FOR aa := 0 TO iSafetyDiag_Anzahl_FbTwoHand DO
	(*	TwoHand (Taster) Diagnose		*)
	fbDiag_TwoHand[aa].stIn := Iarr_SafetyDiag_TwoHand[aa];
	fbDiag_TwoHand[aa]( );
	(*	Warnungen anzeigen	*)
	IF fbDiag_TwoHand[aa].bWarning THEN
		IEvent.Select(Tc_Events.TwinSafeEventClass.ErrorEvent)
			  .ArgSbInitWs(stTextListGlobal.stText_Safety.stText_Safety_FB_Error.wsName)
		  	  .ArgSbAppend(' | ')
			  .ArgSbAppendWsRaise(fbDiag_TwoHand[aa].stWarningText.wsName);
	END_IF
	(*	Error anzeigen	*)
	IF fbDiag_TwoHand[aa].bError THEN
		IEvent.Select(Tc_Events.TwinSafeEventClass.ErrorEvent)
			  .ArgSbInitWs(stTextListGlobal.stText_Safety.stText_Safety_FB_Error.wsName)
		  	  .ArgSbAppend(' | ')
			  .ArgSbAppendWsRaise(fbDiag_TwoHand[aa].stErrorText.wsName);
	END_IF
END_FOR

// EDM Diagnose
FOR aa := 0 TO iSafetyDiag_Anzahl_FbEDM DO
	(*	EDM FB Diagnose		*)
	fbDiag_EDM[aa].stIn := Iarr_SafetyDiag_EDM[aa];
	fbDiag_EDM[aa]( );
	(*	Error anzeigen	*)
	IF fbDiag_EDM[aa].bError THEN
		IEvent.Select(Tc_Events.TwinSafeEventClass.EdmErrorEvent)
			  .ArgSbInitWs(stTextListGlobal.stText_Safety.stText_Safety_FB_Error.wsName)
		  	  .ArgSbAppend(' | ')
			  .ArgSbAppendWsRaise(fbDiag_EDM[aa].stErrorText.wsName);
	END_IF
END_FOR


(*	Hardware	*)
FOR aa := 1 TO iSafety_Anzahl_EL69xx DO
	fbTwinSAFE_HW_Diag[aa].bEnable := Services.bPlcInitDone;
	fbTwinSAFE_HW_Diag[aa].stEcMasterAmsAdr := IO.stControlCabinetIO.stIn.stEtherCATMasterAmsAdr;
	fbTwinSAFE_HW_Diag[aa].nEcMasterDevId := IO.stControlCabinetIO.stIn.uiEcMasterDevId;
	fbTwinSAFE_HW_Diag[aa].nDeviceState := IO.stControlCabinetIO.stIn.eEtherCATDeviceState;
	fbTwinSAFE_HW_Diag[aa].dtNow := Statics.dtNow; // current system time
	fbTwinSAFE_HW_Diag[aa]();
	IF fbTwinSAFE_HW_Diag[aa].bError THEN
		IEvent.Select(Tc_Events.TwinSafeEventClass.HwErrorEvent)
		  	  .ArgSbInitWs(fbTwinSAFE_HW_Diag[aa].stErrorText.wsName)
		  	  .ArgSbAppendRaise(' | Safety Feedback Not-Halt');
	END_IF
END_FOR
END_METHOD

METHOD private M_DoorSequence : BOOL
VAR_INPUT
END_VAR
// Safe Gates

// A
fbSaftyDoors[0].sName := 'Tür Ofen A';
fbSaftyDoors[0].bAblaufGestoppt := Services.stGlobalModuleInfo.bStation_All_Stopped;
fbSaftyDoors[0].bFreigabeTuerEntriegeln := NOT fbSaftyDoors[0].bSAFE_AnforderungSchutzbereich_Ein;
fbSaftyDoors[0](stIO := Safety.arrSaftyDoors[0]);
IF fbSaftyDoors[0].bError THEN
	IEvent.Select(Tc_Events.TwinSafeEventClass.ErrorEvent)
		  .ArgSbInit('Türe A Fehler | ')
		  .ArgSbAppendWsRaise(fbSaftyDoors[0].stErrorText.wsName);
END_IF

// B
fbSaftyDoors[1].sName := 'Tür Ofen B';
fbSaftyDoors[1].bAblaufGestoppt := Services.stGlobalModuleInfo.bStation_All_Stopped;
fbSaftyDoors[1].bFreigabeTuerEntriegeln := NOT fbSaftyDoors[1].bSAFE_AnforderungSchutzbereich_Ein;
fbSaftyDoors[1](stIO := Safety.arrSaftyDoors[1]);
IF fbSaftyDoors[1].bError THEN
	IEvent.Select(Tc_Events.TwinSafeEventClass.ErrorEvent)
		  .ArgSbInit('Türe B Fehler | ')
		  .ArgSbAppendWsRaise(fbSaftyDoors[1].stErrorText.wsName);
END_IF

// reset
rtrigReset(CLK := HMI.stHmi.stIn.stSafety.bQuitSafety);
IF rtrigReset.Q THEN
	FOR ii := 0 TO 1 DO
		fbSaftyDoors[ii].M_Reset();
	END_FOR
END_IF

// request manual on request open door
bMachineRequestCycleStop := NOT (fbSaftyDoors[0].bFreigabeAblauf AND fbSaftyDoors[1].bFreigabeAblauf);
bMachineRequestStart := NOT bMachineRequestCycleStop AND (fbSaftyDoors[0].bStartAblauf OR fbSaftyDoors[1].bStartAblauf);
END_METHOD

METHOD private M_Edm : BOOL
VAR_INPUT
END_VAR
//ToDo: EDM
//bEdm_EmergencyStop:=TRUE;
//stEdm_State_Nothalt:= F_CreateDynText("Alle EDM Nothalt Signale OK", 0);	
//
//stIO.stOut.bSafety_EDM_OUT[E_EDM_Out.eEdmOut_Nothalt] := bEdm_EmergencyStop; //Nothalt

//stIO.stOut.bSafety_EDM_OUT[E_EDM_Out.eEdmOut_Modul1_Freigabeventil] := IO.st001_Modul_IO.stIn.bSignal_Modul1SafetyEdmVentilinsel;//AND IO.st001_Modul_IO.stIn.bSensor_Modul1PilotluftDs;//NOT stIO.stIn.bSafety_Aktor[E_Safety_Actor.eSafety_Actor_Freigabeventil_Area1];

//stIO.stOut.bSafety_EDM_OUT[E_EDM_Out.eEdmOut_Modul1_Rtt] := NOT SafetyArea2_Ok;

//EDM Check Meldungen

//fbEdmCheck[1].bEnable := TRUE;
//fbEdmCheck[1].bActor := stIO.stIn.bSAFE_ES_Ok;
//fbEdmCheck[1].bEdm := stIO.stOut.bSafety_EDM_OUT[E_EDM_Out.eEdmOut_Nothalt];
//fbEdmCheck[1].tActorOnEdmOffDelay := T#1S;
//fbEdmCheck[1].tActorOffEdmOnDelay := T#1S;
//fbEdmCheck[1]();
//IF fbEdmCheck[1].bEdmError THEN
//	fbEdmCheck[1].M_Reset();	
//																		
//	INotiHdl.M_SetNotification(F_CreateDynText("0",0),
//					stTextListGlobal.stText_NG_Safety, 							// Grp
//					stTextListGlobal.stText_Safety.stText_Safety_ES, 			// Text 1 (stTextListGlobal / F_CreateDynText("xxx",0))				 
//					F_CreateDynText("EDM Nothalt",0), 							// Text 2 (stTextListGlobal / F_CreateDynText("xxx",0))
//					stEdm_State_Nothalt,										// Text 3 (stTextListGlobal / F_CreateDynText("xxx",0))	
//					E_AlarmPriority.Warning,									// Priority
//					E_NotificationMode.eNotificationMode_Auto					// Notification mode (Autoreset or manually reset by user)
//					);										
//										
//END_IF
END_METHOD

METHOD private M_General : BOOL
VAR_INPUT
END_VAR
;
//Zustimm bereits in Safety ausgewertet mit Betriebsart
END_METHOD

METHOD INTERNAL M_Init : BOOL
VAR_INPUT
END_VAR
// init Safety stuff here...

// set up logger
ILog := Services.ILog;

// set up safety IOs
stIO REF= IO.stSafetyIO;

// set up event handler 
IEvent := Services.fbEventHandler;

//aSClearText[EN] := 'Safety init done.';
M_Init := TRUE;
END_METHOD

METHOD PRIVATE M_Mapping : BOOL
VAR_INPUT
END_VAR
stIO.stIn.bSAFE_DRIVES_STO := stIO.stIn.bSAFE_DRIVE_A_STO OR
								stIO.stIn.bSAFE_DRIVE_B_STO OR
								stIO.stIn.bSAFE_DRIVES_HG_STO;
								
//IO.stSafetyIO.stIn.bSAFE_Areas_Ok := IO.stSafetyIO.stIn. AND 
//									 IO.stSafetyIO.stIn.bSAFE_Area_Ok_ST20;
									 
									 
// machine stop from safety (ES/Door stop ramp)
bMachineRequestStop := NOT (stIO.stIn.bSAFE_ES_Ok AND
							IO.stSafetyIO.stIn.bSAFE_Areas_Ok );// AND
							//IO.stSafetyIO.stIn.bSAFE_Area_Ok_ST20);
END_METHOD

{attribute 'monitoring' := 'call'}
PROPERTY OpMode_Auto : BOOL
GET
OpMode_Auto := stIO.stIn.bSafe_OpMode_Auto;
END_GET
END_PROPERTY

{attribute 'monitoring' := 'call'}
PROPERTY OpMode_Manual : BOOL
GET
OpMode_Manual := stIO.stIn.bSafe_OpMode_Manual;
END_GET
END_PROPERTY

{attribute 'monitoring' := 'call'}
PROPERTY OpMode_Off : BOOL
GET
OpMode_Off := stIO.stIn.bSafe_OpMode_Off;
END_GET
END_PROPERTY

PROPERTY OpMode_Ruest : BOOL
GET
OpMode_Ruest := stIO.stIn.bSafe_OpMode_Ruest;
END_GET
END_PROPERTY

{attribute 'monitoring' := 'call'}
PROPERTY INTERNAL SafetyAreaOk_ST10 : BOOL
GET
SafetyAreaOk_ST10 := tofAreaOkST10.Q;
END_GET
END_PROPERTY

PROPERTY PUBLIC SafetyAreaOk_ST20 : BOOL
GET
SafetyAreaOk_ST20 := IO.stSafetyIO.stIn.bSAFE_Area_Ok_ST20;
END_GET
END_PROPERTY

{attribute 'monitoring' := 'call'}
PROPERTY PUBLIC SafetyOk : BOOL
GET // PUBLIC
SafetyOk := EmergencyStopOk AND IO.stSafetyIO.stIn.bSAFE_Areas_Ok;
END_GET
END_PROPERTY

END_PROGRAM

// ---- POUs/Safety/Components/Euchner_MGB2/FB_SafeDoorMGB2.TcPOU
FUNCTION_BLOCK FB_SafeDoorMGB2
VAR_IN_OUT
	// IO reference
	stIO 				: ST_MGB2_IO;
END_VAR
VAR_INPUT
	/// Name der Schutztuere
	sName								:STRING;
	
	bEnableSubModul_1					:BOOL := TRUE;
	bEnableSubModul_2					:BOOL := TRUE;
	
	/// Ablauf der Anlage gestoppt -> Freigabe zum Abschalten der Safety
	bAblaufGestoppt						:BOOL;
	
	/// Tuere entriegeln von Safety (Feedbacks)
	bFreigabeTuerEntriegeln				:BOOL;
END_VAR
VAR_OUTPUT
	/// Fehler
	bError								:BOOL;
	stErrorText							:ST_Text;
	
	/// Freigabe an Anlagenbereich zum Ausfueren der Abläufe
	bFreigabeAblauf							:BOOL;
	
	/// Anforderung an Safety für Sicherheit
	bSAFE_AnforderungSchutzbereich_Ein		:BOOL;
END_VAR
VAR
	stInMgb						: ST_Euchner_MGB2_IN;
	stOutMgb					: ST_Euchner_MGB2_Out;
	stInMsm						: ST_Euchner_MSM_IN;
	stOutMsm					: ST_Euchner_MSM_Out;
	stInMsmConfirm				: ST_Euchner_MSM_DA_IN;
	stOutMsmConfirm				: ST_Euchner_MSM_DA_Out;
	
	bReset,
	bStarting,
	bLockDoorRequest,
	bOpenDoorRequest			:BOOL;
	fbTaAnforderung				:FB_TON_RMTH;
	fbTaQuittieren				:FB_TON_RMTH;
	fbSafetyOk					:FB_TON_RMTH;
	tonReset					: TON;
END_VAR

M_Mapping();
M_Supervision();

// Timer, Flanken
fbTaAnforderung(IN := stInMsm.bSM_I_S2, PT:= T#50MS);		// stIO.stIn.bTa_Gelb_S2
fbTaQuittieren(IN := stInMsm.bSM_I_S3, PT:= T#50MS);		// stIO.stIn.bTa_Weiss_S3

stOutMsm.bSM_O_H1 := FALSE;
stOutMsm.bSM_O_H2 := FALSE;
stOutMsm.bSM_O_H3 := FALSE;

tonReset.IN := bReset;
tonReset.PT := T#150MS;
tonReset();
IF tonReset.Q THEN
	bReset := FALSE;
END_IF
stOutMgb.bLM_ACK_ER := stOutMgb.bLM_ACK_G := bReset;
stOutMgb.bLM_ACK_G := stOutMgb.bLM_ACK_G := bReset;

(*	Funktion OK	*)
IF NOT bError THEN

	// mapp ES button to led
	IF NOT stInMsm.bSM_I_S1 THEN
		stOutMsm.bSM_O_H1 := Statics.stPulse.bToggle500ms; 
	ELSE
		stOutMsm.bSM_O_H1 := FALSE;
	END_IF

	//---------------------------- Open ---------------------------------
	// Anforderung Tuere oeffnen
	IF fbTaAnforderung.Qr OR bOpenDoorRequest THEN
		bOpenDoorRequest := FALSE;
		bFreigabeAblauf := FALSE;
		bStarting := FALSE;
	END_IF
	// Safety abschalten
	IF NOT bFreigabeAblauf AND bAblaufGestoppt AND 	// Abläufe sind gestoppt in dem Bereich
	NOT bStarting THEN
		bSAFE_AnforderungSchutzbereich_Ein := FALSE;		// Abschalten in Safety
	END_IF
	
	// Rückmeldung von Safety das entriegelt werden darf
	IF NOT bSAFE_AnforderungSchutzbereich_Ein AND 
	bFreigabeTuerEntriegeln AND NOT bStarting THEN
		stOutMgb.bLM_O_CL := TRUE; // entriegeln	
	END_IF
	
	
	// Signal LED - Gelb
	IF bStarting THEN
		stOutMsm.bSM_O_H2 := FALSE;	
	ELSIF NOT bFreigabeAblauf AND NOT bFreigabeTuerEntriegeln THEN
		stOutMsm.bSM_O_H2 := Statics.stPulse.bToggle500ms;
	ELSIF NOT stIO.bSAFE_DoorSafetyOk THEN
		stOutMsm.bSM_O_H2 := TRUE;
	ELSE
		stOutMsm.bSM_O_H2 := FALSE;
	END_IF
	
	
	//---------------------------- Close + Start --------------------------
	// Tuere quittieren (geschlossen und verriegeln) -> fallende Flanke
	IF fbTaQuittieren.Qf OR bLockDoorRequest THEN
		bLockDoorRequest := FALSE;
		IF stInMgb.bLM_I_SK AND stInMgb.bLM_I_OL THEN	// stIO.stIn.bMeldungRiegelzunge_OT   stInMgb.bLM_I_SK AND stInMgb.bLM_I_OL
			stOutMgb.bLM_O_CL := FALSE; // verriegeln
			bSAFE_AnforderungSchutzbereich_Ein := TRUE;	// Safety Ein
			bStarting := TRUE;
		END_IF
	END_IF
	
	fbSafetyOk(IN := stIO.bSAFE_DoorSafetyOk, PT := T#200MS);
	IF bStarting THEN
		IF fbSafetyOk.Q THEN
			bFreigabeAblauf := TRUE;
			bStarting := FALSE;
		END_IF
	END_IF
	
	// Signal LED - Weiss
	IF stIO.bSAFE_DoorSafetyOk THEN
		stOutMsm.bSM_O_H3 := TRUE;
	ELSIF bStarting THEN
		stOutMsm.bSM_O_H3 := Statics.stPulse.bToggle500ms;
	ELSIF stInMgb.bLM_I_OT THEN		// stIO.stIn.bMeldungRiegelzunge_OT
		stOutMsm.bSM_O_H3 := Statics.stPulse.bToggle1000ms;
	ELSE
		stOutMsm.bSM_O_H3 := FALSE;
	END_IF
	
// 
// ERROR
ELSE

	stOutMsm.bSM_O_H1 := Statics.stPulse.bToggle500ms;
	stOutMsm.bSM_O_H2 := Statics.stPulse.bToggle500ms;
	stOutMsm.bSM_O_H3 := Statics.stPulse.bToggle500ms;

	stOutMgb.bLM_O_CL := TRUE;
	IF stInMsm.bSM_I_S2 OR stInMsm.bSM_I_S3 THEN
		bReset := TRUE;
	END_IF
	IF stInMsm.bSM_I_S2 AND stInMgb.bLM_I_SK AND stInMgb.bLM_I_OL THEN
		stOutMgb.bLM_O_CL := FALSE;
	ELSIF stInMsm.bSM_I_S3 THEN	(*AND bEnable*)
		stOutMgb.bLM_O_CL := TRUE;
	END_IF
	
END_IF

stIO.bSAFE_UnlockDoor := stOutMgb.bLM_O_CL;

METHOD PRIVATE M_Error : BOOL
VAR_INPUT
	stError: ST_Text;
END_VAR
bError	:=TRUE;
stErrorText	:= stError;
END_METHOD

METHOD M_LockDoor : BOOL
VAR_INPUT
END_VAR
//IF stInMgb.bLM_I_OT THEN
	bLockDoorRequest := TRUE;	
//END_IF
END_METHOD

METHOD PRIVATE M_Mapping : BOOL
//mgb mapping in
stInMgb.bLM_D_RUN := 	stIO.stHwInMgb.nByte0.0;
stInMgb.bLM_I_SK := 	stIO.stHwInMgb.nByte0.1;
stInMgb.bLM_E_SM1 := 	stIO.stHwInMgb.nByte0.2;
stInMgb.bLM_E_SM2 := 	stIO.stHwInMgb.nByte0.3;
stInMgb.bLM_E_ER := 	stIO.stHwInMgb.nByte0.4;
stInMgb.bLM_E_G := 		stIO.stHwInMgb.nByte0.5;
stInMgb.bLM_I_OD := 	stIO.stHwInMgb.nByte0.6;
stInMgb.bLM_I_OT := 	stIO.stHwInMgb.nByte0.7;
stInMgb.bLM_I_OL := 	stIO.stHwInMgb.nByte1.0;

//mgb mapping out
stIO.stHwOutMgb.nByte0.0 := stOutMgb.bLM_O_CL;
stIO.stHwOutMgb.nByte0.1 := stOutMgb.bLM_ACK_ER;
stIO.stHwOutMgb.nByte0.2 := stOutMgb.bLM_ACK_G;

//msm mapping in
stInMsm.bSM_I_S1 := 	stIO.stHwInMsm.nByte0.0;
stInMsm.bSM_I_S2 := 	stIO.stHwInMsm.nByte0.1;
stInMsm.bSM_I_S3 := 	stIO.stHwInMsm.nByte0.2;
stInMsm.bSM_E_S1 := 	stIO.stHwInMsm.nByte0.5;

stInMsmConfirm.bSM_I_X3 := 	stIO.stHwInMsmConfirm.nByte0.0;	// Zustimm
stInMsmConfirm.bSM_I_T1 := 	stIO.stHwInMsmConfirm.nByte0.2;	// Minus
stInMsmConfirm.bSM_I_T2 := 	stIO.stHwInMsmConfirm.nByte0.1; // Plus
stInMsmConfirm.bSM_E_X3 := 	stIO.stHwInMsmConfirm.nByte0.5;

//msm mapping out
stIO.stHwOutMsm.nByte0.0 := stOutMsm.bSM_O_H1;
stIO.stHwOutMsm.nByte0.1 := stOutMsm.bSM_O_H2;
stIO.stHwOutMsm.nByte0.2 := stOutMsm.bSM_O_H3;
stIO.stHwOutMsm.nByte0.3 := stOutMsm.bSM_O_H1_B;
stIO.stHwOutMsm.nByte0.4 := stOutMsm.bSM_O_H2_B;
stIO.stHwOutMsm.nByte0.5 := stOutMsm.bSM_O_H3_B;

stIO.stHwOutMsmConfirm.nByte0.0 := stOutMsmConfirm.bSM_O_L2;
stIO.stHwOutMsmConfirm.nByte0.1 := stOutMsmConfirm.bSM_O_L1;
stIO.stHwOutMsmConfirm.nByte0.3 := stOutMsmConfirm.bSM_O_L2_B;
stIO.stHwOutMsmConfirm.nByte0.4 := stOutMsmConfirm.bSM_O_L1_B;
END_METHOD

METHOD M_OpenDoor : BOOL
VAR_INPUT
END_VAR
bOpenDoorRequest := TRUE;
END_METHOD

METHOD M_Reset : BOOL
bReset	:= TRUE;
bError	:= FALSE;
MEMSET(ADR(stErrorText),0,SIZEOF(stErrorText));
END_METHOD

METHOD PRIVATE M_Supervision : BOOL
IF stInMgb.bLM_E_SM1 AND bEnableSubModul_1 AND FALSE THEN
	M_Error(F_CreateDynTextEx(0, "Safety_MGB2_ErrBit_Submod1", "MGB2 - Fehlermeldebit für Submodul 1")); 	
ELSIF stInMgb.bLM_E_SM2 AND bEnableSubModul_2 THEN
	M_Error(F_CreateDynTextEx(0, "Safety_MGB2_ErrBit_Submod2", "MGB2 - Fehlermeldebit für Submodul 2"));	
ELSIF stInMgb.bLM_E_ER THEN
	M_Error(F_CreateDynTextEx(0, "Safety_MGB2_ErrBit_EscapeUnlock", "MGB2 - für Fluchtentriegelung"));	
ELSIF stInMgb.bLM_E_G THEN
	M_Error(F_CreateDynTextEx(0, "Safety_MGB2_ErrBit_ModError", "MGB2 - allgemeiner Modulfehler"));
ELSIF stInMsm.bSM_E_S1 THEN
	M_Error(F_CreateDynTextEx(0, "Safety_MSM_ErrBit_Sx", "MSM - Fehler"));
END_IF
END_METHOD

END_FUNCTION_BLOCK

// ---- POUs/HMI/Utilities/DynTxt/F_CreateDynTextEx.TcPOU
FUNCTION F_CreateDynTextEx : ST_Text
VAR_INPUT
	nNameId		: INT;		//example simatic hmi
	wsNameId	: WSTRING;	//standard name
	wsName		: WSTRING;	//standard name
END_VAR

F_CreateDynTextEx.nNameId := nNameId;
F_CreateDynTextEx.wsNameId := wsNameId;
F_CreateDynTextEx.wsName := wsName;

END_FUNCTION

// ---- POUs/Safety/Components/SafetyDoor/FB_SafetyDoor.TcPOU
FUNCTION_BLOCK FB_SafetyDoor
VAR_IN_OUT
	// IO reference
	stIO 				: ST_SafetyDoor_IO;
END_VAR
VAR_INPUT
	/// Name der Schutztuere
	sName								:STRING;
	
	bEnableSubModul_1					:BOOL := TRUE;
	bEnableSubModul_2					:BOOL := TRUE;
	
	/// Ablauf der Anlage gestoppt -> Freigabe zum Abschalten der Safety
	bAblaufGestoppt						:BOOL;
	
	/// Tuere entriegeln von Safety (Feedbacks)
	bFreigabeTuerEntriegeln				:BOOL;
END_VAR
VAR_OUTPUT
	/// Fehler
	bError								:BOOL;
	stErrorText							:ST_Text;
	
	/// Freigabe an Anlagenbereich zum Ausfueren der Abläufe
	bFreigabeAblauf,
	bStartAblauf 						: BOOL;
	
	/// Anforderung an Safety für Sicherheit
	bSAFE_AnforderungSchutzbereich_Ein	: BOOL;
END_VAR
VAR
	stIn					: ST_SafetyDoor_IN;
	stOut					: ST_SafetyDoor_OUT;
	
	bReset,
	bStarting				: BOOL;
	fbTaAnforderung			:FB_TON_RMTH;
	fbTaLock				:FB_TON_RMTH;
	fbTaStart				:FB_TON_RMTH;
	fbSafetyOk				:FB_TON_RMTH;
	tonReset, tonDelay		: TON;
	nStep					: INT;
END_VAR

M_Mapping();

// Timer, Flanken
fbTaAnforderung(IN := stIn.bRequestButton, PT:= T#50MS);	//Blau	
fbTaLock(IN := stIn.bLockButton, PT:= T#50MS);				//Gelb 
fbTaStart(IN := stIn.bStartButton, PT:= T#50MS);			//Grün 
fbSafetyOk(IN := stIn.tsSafe, PT := T#200MS);				//Safety

bStartAblauf := FALSE;

tonReset.IN := bReset;
tonReset.PT := T#150MS;
tonReset();
IF tonReset.Q THEN
	bReset := FALSE;
END_IF
//stOut.tsRestart := bReset;

(*	Funktion OK	*)
IF NOT bError THEN

	//---------------------------- Open ---------------------------------
	// Anforderung Tuere oeffnen
	IF fbTaAnforderung.Qr THEN
		bFreigabeAblauf := FALSE;
		bStarting := FALSE;
	END_IF
	
	// Safety abschalten
	IF NOT bFreigabeAblauf AND bAblaufGestoppt AND 	 // Abläufe sind gestoppt in dem Bereich
	NOT bStarting THEN
		bSAFE_AnforderungSchutzbereich_Ein := FALSE; // Abschalten in Safety
	END_IF
	
	// Rückmeldung von Safety das entriegelt werden darf
	IF fbTaLock.Qf THEN
		//---------------------------- Close + Start --------------------------
		// Tuere quittieren (geschlossen und verriegeln) -> fallende Flanke
		IF NOT stOut.tsLockCmd THEN
			nStep := 10; // lock
		ELSE
			nStep := 100; // open
		END_IF
	END_IF
	
	IF fbTaStart.Qf OR bStarting THEN
		IF fbSafetyOk.Q THEN
			bFreigabeAblauf := TRUE;
			bStartAblauf := TRUE;
			bStarting := FALSE;
		END_IF
	END_IF
	
	
	
	//---------------------------- Lights --------------------------	
	// Signal LED - Grün/Gelb	
	IF Services.stGlobalModuleInfo.bStation_All_Auto THEN
		IF Services.stGlobalModuleInfo.bStation_All_Started THEN
			stOut.bStartLight := TRUE;
			stOut.bStopLight := FALSE;
		ELSIF Services.stGlobalModuleInfo.bStation_All_Stopped THEN
			stOut.bStartLight := FALSE;
			stOut.bStopLight := TRUE;
		ELSIF bFreigabeAblauf THEN
			stOut.bStartLight := Statics.stPulse.bToggle500ms;
			stOut.bStopLight := Statics.stPulse.bToggle500ms;
		END_IF
	ELSE
		stOut.bStartLight := FALSE;
		stOut.bStopLight := FALSE;
	END_IF	
	
	// Signal LED - Gelb
	stOut.bLockLight := NOT stIn.tsOpen;	
// 
// ERROR
ELSE

	stOut.bLockLight := Statics.stPulse.bToggle500ms;
	stOut.bStopLight := Statics.stPulse.bToggle500ms;
	stOut.tsLockCmd := FALSE;
	
END_IF

tonDelay();
CASE nStep OF
	0: // idle
		IF stIn.tsOpen THEN
			nStep := 10;
		END_IF
	
	10: // lock
		IF stIn.tsSafe THEN
			nStep := 30;
		ELSE
			tonDelay(IN := FALSE);
			stOut.tsRestart := TRUE;
			nStep := 20;
		END_IF
		
	20: // restart door fb (delay)
		tonDelay(IN := TRUE, PT := T#300MS);
		IF tonDelay.Q THEN
			tonDelay(IN := FALSE);
			stOut.tsRestart := FALSE;
			nStep := 10;
		END_IF
		
	30: // lock
		stOut.tsLockCmd := TRUE; // verriegeln
		bSAFE_AnforderungSchutzbereich_Ein := TRUE;	// Safety Ein
		bStarting := TRUE;
		nStep := 0;
		
	100: // open
		bFreigabeAblauf := FALSE;
		bStarting := FALSE;
	
		IF NOT bSAFE_AnforderungSchutzbereich_Ein AND 
		bFreigabeTuerEntriegeln AND NOT bStarting THEN
			stOut.tsLockCmd := FALSE; // entriegeln
			nStep := 0;
		END_IF
		
		
END_CASE

METHOD PRIVATE M_Error : BOOL
VAR_INPUT
	stError: ST_Text;
END_VAR
bError	:=TRUE;
stErrorText	:= stError;
END_METHOD

METHOD PRIVATE M_Mapping : BOOL
//mgb mapping in
stIn := stIO.stHwIn;

stOut.tsLocked := stIn.bLocked;

stIO.stHwOut := stOut;
END_METHOD

METHOD M_Reset : BOOL
bReset	:= TRUE;
bError	:= FALSE;
MEMSET(ADR(stErrorText),0,SIZEOF(stErrorText));
END_METHOD

END_FUNCTION_BLOCK

// ---- POUs/HMI/Utilities/DynTxt/F_CreateDynText.TcPOU
FUNCTION F_CreateDynText : ST_Text
VAR_INPUT
	wsName		: WSTRING;	//standard name
	nNameId		: INT;		//example simatic hmi
END_VAR
VAR
END_VAR

F_CreateDynText.wsName := wsName;
F_CreateDynText.wsNameId := wsName;
F_CreateDynText.nNameId := nNameId;

END_FUNCTION

// ---- POUs/HMI/P_HMI_Controller.TcPOU
/// HMI access provider (host for sub hmi provider)
PROGRAM INTERNAL P_HMI_Controller
VAR_OUTPUT	
	// default items from HMI to module & stations
	aStHmiToModule	: ARRAY[0..E_Module.eModule_nMaxIdx] OF ST_DefaultHmiToPlc;
	aStHmiToStation	: ARRAY[0..E_Station.eStation_nMaxIdx] OF ST_DefaultHmiToPlc;
	bLedTest 		: BOOL;
END_VAR
VAR
	stHmiBaseOut	: ST_HMI_BASE_OUT;
	IEvent			: I_EventHandler;
	aiHmiProvider	: ARRAY[0..E_HMI_PROVIDER.eHmiProvider_nMaxIdx] OF ITF_HMI_PROVIDER;

	// default trigger
	aFbProviderRequestTrigger	: ARRAY[0..E_HMI_PROVIDER.eHmiProvider_nMaxIdx] OF FB_ProviderRequestTrigger;
	
	aFbTrigHmiToModule			: ARRAY[0..eModule_nMaxIdx] OF FB_HmiBaseControlTrigger;
	aFbTrigHmiToStation			: ARRAY[0..eStation_nMaxIdx] OF FB_HmiBaseControlTrigger;
			
	/// private variabe
	ii							: INT;
	stHmiInEmpty 				: ST_HMI_IN;	
	
	sChanges					: T_MaxString;
	fbSettingsHandling 			: FB_SettingsHandling;
	fbMonitoringHandling		: FB_MonitoringHandling;
	
	tonUserLevelLogOut				: TON;
	rTrigUserManagmentLogIn,
	rTrigUserManagmentLogOut,
	rTrigUserManagmentSubmit		: R_TRIG;	
	fTrigUserManagmentSubmit		: F_TRIG;
	rTrigUserManagmentDelete		: R_TRIG;
	
	nUserManagemenetColumnIdx_Old	: UINT;
	nUserManagemenetRowIdx_Old		: UINT;
	
	sUserLevelLastUser				: STRING;
	stAxisManagerDummy 				: ST_AxisManager;
END_VAR
VAR PERSISTENT
	// user data
	iUserLevel					: INT;	(*user level 0 = none 1= Operator 2 = Plant Manager 3 = maintenance 4 = reserve 5= admin 6= programmer*)
	stUserLevel					: ARRAY [0..20] OF ST_User_Management;
	bPasswordSave				: BOOL;
END_VAR

///
/// HMI access provider
/// 

// build general HMI out
M_PlcToHmi();

// init summary IN (resets combined or-signals)
stHMI.stIn := stHmiInEmpty;

// loop provider, run & chk control requests
FOR ii := 0 TO E_HMI_PROVIDER.eHmiProvider_nMaxIdx DO
	IF aiHmiProvider[ii] = 0 THEN CONTINUE;	END_IF
	
	M_PlcToProvider(aiHmiProvider[ii]);
	aiHmiProvider[ii].M_Run();
	IF aiHmiProvider[ii].Mute THEN CONTINUE; END_IF
	M_ProviderToPlc(aiHmiProvider[ii], aFbProviderRequestTrigger[ii]);
END_FOR

bLedTest := stHmi.stIn.stSpecial.stButton_LedTest.bClick;

// build module & station signals
M_HmiToModules();
M_HmiToStations();

// user mgmt --> switched to Beckhoff HMI UserMgmt
HMI.eUserLevel := HMI.stHmiTc3.stIn.stUserMgmt.iHmiUserLevel;
//M_UserManagement();
M_AxisManagement();

// reset
IF stHmi.stIn.stMain.stButton_Reset.bClick THEN
	M_Reset();
END_IF

METHOD PRIVATE M_AddSystemInfo : BOOL
VAR
	idx : INT;
END_VAR
// add/update system infos
idx := 0;
M_UpdateSystemInfo('App.ProjectName', Statics.stPlcSystemInfo.stPlcAppSystemInfo.ProjectName, idx);
M_UpdateSystemInfo('Software Version', stLibVersion_PLC.sVersion, idx);
M_UpdateSystemInfo('Safety Device Serial', UDINT_TO_STRING(IO.stSafetyIO.stIn.nSerialNumber), idx);
M_UpdateSystemInfo('Safety Project CRC', WORD_TO_STRING(IO.stSafetyIO.stIn.nProjectCrc), idx);
M_UpdateSystemInfo('', '', idx);
M_UpdateSystemInfo('App.AppName', Statics.stPlcSystemInfo.stPlcAppSystemInfo.AppName, idx);
M_UpdateSystemInfo('App.AppTimestamp', DT_TO_STRING(Statics.stPlcSystemInfo.stPlcAppSystemInfo.AppTimestamp), idx);
M_UpdateSystemInfo('App.AdsPort', UDINT_TO_STRING(Statics.stPlcSystemInfo.stPlcAppSystemInfo.AdsPort), idx);
M_UpdateSystemInfo('App.ObjId', UDINT_TO_STRING(Statics.stPlcSystemInfo.stPlcAppSystemInfo.ObjId), idx);
M_UpdateSystemInfo('App.TaskCnt', UDINT_TO_STRING(Statics.stPlcSystemInfo.stPlcAppSystemInfo.TaskCnt), idx);
M_UpdateSystemInfo('App.OnlineChangeCnt', UDINT_TO_STRING(Statics.stPlcSystemInfo.stPlcAppSystemInfo.OnlineChangeCnt), idx);
M_UpdateSystemInfo('App.Flags', DWORD_TO_STRING(Statics.stPlcSystemInfo.stPlcAppSystemInfo.Flags), idx);
M_UpdateSystemInfo('App.BootDataLoaded', BOOL_TO_STRING(Statics.stPlcSystemInfo.stPlcAppSystemInfo.BootDataLoaded), idx);
M_UpdateSystemInfo('App.OldBootData', BOOL_TO_STRING(Statics.stPlcSystemInfo.stPlcAppSystemInfo.OldBootData), idx);
M_UpdateSystemInfo('App.KeepOutputsOnBP', BOOL_TO_STRING(Statics.stPlcSystemInfo.stPlcAppSystemInfo.KeepOutputsOnBP), idx);
M_UpdateSystemInfo('App.ShutdownInProgress',  BOOL_TO_STRING(Statics.stPlcSystemInfo.stPlcAppSystemInfo.ShutdownInProgress), idx);
M_UpdateSystemInfo('App.LicensesPending',  BOOL_TO_STRING(Statics.stPlcSystemInfo.stPlcAppSystemInfo.LicensesPending), idx);
M_UpdateSystemInfo('App.BSODOccured',  BOOL_TO_STRING(Statics.stPlcSystemInfo.stPlcAppSystemInfo.BSODOccured), idx);	 
//M_AddSystemInfo('App.TComSrvPtr', Statics.stPlcSystemInfo.stPlcAppSystemInfo.TComSrvPtr, idx); 
M_UpdateSystemInfo('Task.TaskName', Statics.stPlcSystemInfo.stPlcTaskSystemInfo.TaskName, idx);
M_UpdateSystemInfo('Task.AdsPort', UINT_TO_STRING(Statics.stPlcSystemInfo.stPlcTaskSystemInfo.AdsPort), idx);
M_UpdateSystemInfo('Task.Priority', UINT_TO_STRING(Statics.stPlcSystemInfo.stPlcTaskSystemInfo.Priority), idx);
M_UpdateSystemInfo('Task.CycleTime', Concat2x(F_LRealToStringEx(Statics.stPlcSystemInfo.fCycleTime * 1E3, 0), ' ms, '), idx);
M_UpdateSystemInfo('Task.LastExecTime', Concat2x(F_LRealToStringEx(Statics.stPlcSystemInfo.fLastExecTime * 1E6, 1), ' µs'), idx);
M_UpdateSystemInfo('Task.CycleCount',UDINT_TO_STRING(Statics.stPlcSystemInfo.stPlcTaskSystemInfo.CycleCount), idx);
M_UpdateSystemInfo('Task.DcTaskTime', LINT_TO_STRING(Statics.stPlcSystemInfo.stPlcTaskSystemInfo.DcTaskTime), idx);
M_UpdateSystemInfo('Task.FirstCycle', BOOL_TO_STRING(Statics.stPlcSystemInfo.stPlcTaskSystemInfo.FirstCycle), idx);
M_UpdateSystemInfo('Task.CycleTimeExceeded', BOOL_TO_STRING(Statics.stPlcSystemInfo.stPlcTaskSystemInfo.CycleTimeExceeded), idx);
M_UpdateSystemInfo('Task.InCallAfterOutputUpdate', BOOL_TO_STRING(Statics.stPlcSystemInfo.stPlcTaskSystemInfo.InCallAfterOutputUpdate), idx);
M_UpdateSystemInfo('Task.RTViolation', BOOL_TO_STRING(Statics.stPlcSystemInfo.stPlcTaskSystemInfo.RTViolation), idx);
END_METHOD

METHOD M_AxisManagement : INT
VAR_INPUT
	
END_VAR
IF NOT Services.bPlcInitDone THEN
	RETURN;
END_IF

HMI.stHmiInOut.stHmiAxisManager.bEnableAxisMgr := P_Safety.OpMode_Off;

CASE HMI.stHmiInOut.stHmiAxisManager.eAxis OF
	E_Axis.eAxis_OvenA: HMI.stHmiInOut.stHmiAxisManager.stAxisManager REF= fbSt010OvenA.fbAxisUi.stAxisManager;
	E_Axis.eAxis_OvenB: HMI.stHmiInOut.stHmiAxisManager.stAxisManager REF= fbSt020OvenB.fbAxisUi.stAxisManager;
	
	E_Axis.eAxis_Handling_X: HMI.stHmiInOut.stHmiAxisManager.stAxisManager REF= fbSt030Handling.fbAxisXUi.stAxisManager;
	E_Axis.eAxis_Handling_Y: HMI.stHmiInOut.stHmiAxisManager.stAxisManager REF= fbSt030Handling.fbAxisYUi.stAxisManager;
	E_Axis.eAxis_Handling_Z: HMI.stHmiInOut.stHmiAxisManager.stAxisManager REF= fbSt030Handling.fbAxisZUi.stAxisManager;
	
	ELSE
		;//HMI.stHmiInOut.stHmiAxisManager.stAxisManager REF= fbModul001.fbAxisVmUi.stAxisManager;
END_CASE
END_METHOD

METHOD PRIVATE M_CombineCommonSignals : BOOL
VAR_IN_OUT
	stCtrlSum : ST_HMI_BASE_CONTROL_IN;
	stCtrlPrv : ST_HMI_BASE_CONTROL_IN;
END_VAR
F_OR_REF(stCtrlSum.stButton_Start.bClick, 		stCtrlPrv.stButton_Start.bClick);
F_OR_REF(stCtrlSum.stButton_CycleStop.bClick,	stCtrlPrv.stButton_CycleStop.bClick);
F_OR_REF(stCtrlSum.stButton_Stop.bClick, 		stCtrlPrv.stButton_Stop.bClick);
F_OR_REF(stCtrlSum.stButton_Home.bClick, 		stCtrlPrv.stButton_Home.bClick);
F_OR_REF(stCtrlSum.stButton_Step.bClick, 		stCtrlPrv.stButton_Step.bClick);
F_OR_REF(stCtrlSum.stButton_Reset.bClick, 		stCtrlPrv.stButton_Reset.bClick);
F_OR_REF(stCtrlSum.stButton_OPM_Auto.bClick,	stCtrlPrv.stButton_OPM_Auto.bClick);
F_OR_REF(stCtrlSum.stButton_OPM_Step.bClick,	stCtrlPrv.stButton_OPM_Step.bClick);
F_OR_REF(stCtrlSum.stButton_OPM_Manual.bClick,	stCtrlPrv.stButton_OPM_Manual.bClick);

M_CombineCommonSignals := TRUE;
END_METHOD

METHOD PRIVATE M_HmiToModules : BOOL
VAR
	ii	: INT;
END_VAR
// loop modules, default HMI to module (start, stop, reset, OpModes,...)
FOR ii := 0 TO E_Module.eModule_nMaxIdx DO
	// run only for valid modules
	IF P_Plant.aIModule[ii] = 0 THEN
		CONTINUE;
	END_IF

	aFbTrigHmiToModule[ii].stHmiToPlcIn.bStart := 			stHmi.stIn.arrStModule[ii].stButton_Start.bClick OR 
															stHmi.stIn.stMain.stButton_Start.bClick;
															
	aFbTrigHmiToModule[ii].stHmiToPlcIn.bStop := 			stHmi.stIn.arrStModule[ii].stButton_CycleStop.bClick OR 
															stHmi.stIn.stMain.stButton_Stop.bClick;
															
	aFbTrigHmiToModule[ii].stHmiToPlcIn.bFastStop := 		stHmi.stIn.arrStModule[ii].stButton_Stop.bClick OR 
															stHmi.stIn.stMain.stButton_CycleStop.bClick;
															
	aFbTrigHmiToModule[ii].stHmiToPlcIn.bReset := 			stHmi.stIn.arrStModule[ii].stButton_Reset.bClick OR 
															stHmi.stIn.stMain.stButton_Reset.bClick;

	aFbTrigHmiToModule[ii].stHmiToPlcIn.bStep := 			stHmi.stIn.arrStModule[ii].stButton_Step.bClick OR 
															stHmi.stIn.stMain.stButton_Step.bClick; 
															
	aFbTrigHmiToModule[ii].stHmiToPlcIn.bHome := 			stHmi.stIn.arrStModule[ii].stButton_Home.bClick OR 
															stHmi.stIn.stMain.stButton_Home.bClick; 
															
	aFbTrigHmiToModule[ii].stHmiToPlcIn.bOpModeManual := 	stHmi.stIn.arrStModule[ii].stButton_OPM_Manual.bClick OR 
															stHmi.stIn.stMain.stButton_OPM_Manual.bClick; 
															
	aFbTrigHmiToModule[ii].stHmiToPlcIn.bOpModeAuto := 		stHmi.stIn.arrStModule[ii].stButton_OPM_Auto.bClick OR 
															stHmi.stIn.stMain.stButton_OPM_Auto.bClick; 
															
	aFbTrigHmiToModule[ii].stHmiToPlcIn.bOpModeStep := 		stHmi.stIn.arrStModule[ii].stButton_OPM_Step.bClick OR 
															stHmi.stIn.stMain.stButton_OPM_Step.bClick;

	IF P_Safety.OpMode_Auto THEN
		aFbTrigHmiToModule[ii].stHmiToPlcIn.eSafetyOpMode := E_OpMode.eOpMode_auto;
	ELSIF P_Safety.OpMode_Manual THEN		
		aFbTrigHmiToModule[ii].stHmiToPlcIn.eSafetyOpMode := E_OpMode.eOpMode_manual;
//		ELSIF P_Safety.Betriebsart_Ruest THEN		
//			aFbTrigHmiToModule[ii].stHmiToPlcIn.eSafetyOpMode := E_OpMode.eOpMode_manual;
	ELSIF P_Safety.OpMode_Off THEN
		aFbTrigHmiToModule[ii].stHmiToPlcIn.eSafetyOpMode := E_OpMode.eOpMode_off;
	ELSE
		aFbTrigHmiToModule[ii].stHmiToPlcIn.eSafetyOpMode := E_OpMode.eOpMode_off;
	END_IF

	aFbTrigHmiToModule[ii](stHmiToPlcOut := aStHmiToModule[ii]);
END_FOR
END_METHOD

METHOD PRIVATE M_HmiToStations : BOOL
VAR
	ii	: INT;
	ISt	: IStation;
END_VAR
// loop stations, default HMI to mostationdule (start, stop, reset, OpModes,...)
FOR ii := 0 TO E_Station.eStation_nMaxIdx DO
	// run only for valid stations
	IF P_Plant.aIStaton[ii] = 0 THEN
		CONTINUE;
	END_IF

	ISt := P_Plant.aIStaton[ii];
	aFbTrigHmiToStation[ii].stHmiToPlcIn.bStart := 			stHmi.stIn.arrStStation[ii].stButton_Start.bClick OR 
															//to start all stations of the module:
															//stHmi.stIn.arrStModule[ISt.Parent].stButton_Start.bClick OR 
															stHmi.stIn.stMain.stButton_Start.bClick;
															
	aFbTrigHmiToStation[ii].stHmiToPlcIn.bStop := 			stHmi.stIn.arrStStation[ii].stButton_CycleStop.bClick OR 
															//stHmi.stIn.arrStModule[ISt.Parent].stButton_CycleStop.bClick OR 
															stHmi.stIn.stMain.stButton_Stop.bClick;
															
	aFbTrigHmiToStation[ii].stHmiToPlcIn.bFastStop := 		stHmi.stIn.arrStStation[ii].stButton_Stop.bClick OR 
															//stHmi.stIn.arrStModule[ISt.Parent].stButton_Stop.bClick OR 
															stHmi.stIn.stMain.stButton_CycleStop.bClick;
															
	aFbTrigHmiToStation[ii].stHmiToPlcIn.bReset := 			stHmi.stIn.arrStStation[ii].stButton_Reset.bClick OR 
															//stHmi.stIn.arrStModule[ISt.Parent].stButton_Reset.bClick OR 
															stHmi.stIn.stMain.stButton_Reset.bClick;

	aFbTrigHmiToStation[ii].stHmiToPlcIn.bStep := 			stHmi.stIn.arrStStation[ii].stButton_Step.bClick OR 
															//stHmi.stIn.arrStModule[ISt.Parent].stButton_Step.bClick OR 
															stHmi.stIn.stMain.stButton_Step.bClick; 
															
	aFbTrigHmiToStation[ii].stHmiToPlcIn.bHome := 			stHmi.stIn.arrStStation[ii].stButton_Home.bClick OR 
															//stHmi.stIn.arrStModule[ISt.Parent].stButton_Home.bClick OR 
															stHmi.stIn.stMain.stButton_Home.bClick; 
															
	aFbTrigHmiToStation[ii].stHmiToPlcIn.bOpModeManual := 	stHmi.stIn.arrStStation[ii].stButton_OPM_Manual.bClick OR 
															//stHmi.stIn.arrStModule[ISt.Parent].stButton_OPM_Manual.bClick OR 
															stHmi.stIn.stMain.stButton_OPM_Manual.bClick; 
															
	aFbTrigHmiToStation[ii].stHmiToPlcIn.bOpModeAuto := 	stHmi.stIn.arrStStation[ii].stButton_OPM_Auto.bClick OR 
															//stHmi.stIn.arrStModule[ISt.Parent].stButton_OPM_Auto.bClick OR 
															stHmi.stIn.stMain.stButton_OPM_Auto.bClick; 
															
	aFbTrigHmiToStation[ii].stHmiToPlcIn.bOpModeStep := 	stHmi.stIn.arrStStation[ii].stButton_OPM_Step.bClick OR 
															//stHmi.stIn.arrStModule[ISt.Parent].stButton_OPM_Step.bClick OR 
															stHmi.stIn.stMain.stButton_OPM_Step.bClick;

	IF P_Safety.OpMode_Auto THEN
		aFbTrigHmiToStation[ii].stHmiToPlcIn.eSafetyOpMode := E_OpMode.eOpMode_auto;
	ELSIF P_Safety.OpMode_Manual THEN		
		aFbTrigHmiToStation[ii].stHmiToPlcIn.eSafetyOpMode := E_OpMode.eOpMode_manual;
//		ELSIF P_Safety.Betriebsart_Ruest THEN		
//			aFbTrigHmiToStation[ii].stHmiToPlcIn.eSafetyOpMode := E_OpMode.eOpMode_manual;
	ELSIF P_Safety.OpMode_Off THEN
		aFbTrigHmiToStation[ii].stHmiToPlcIn.eSafetyOpMode := E_OpMode.eOpMode_off;
	ELSE
		aFbTrigHmiToStation[ii].stHmiToPlcIn.eSafetyOpMode := E_OpMode.eOpMode_off;
	END_IF

	aFbTrigHmiToStation[ii](stHmiToPlcOut := aStHmiToStation[ii]);
END_FOR
END_METHOD

METHOD INTERNAL M_Init : BOOL
VAR_INPUT
END_VAR
VAR
	nn : INT;
END_VAR
//aSClearText[EN] := 'Initialize HMI';

// set up defaults
M_SetReferences(Services.fbEventHandler);

// init HMI stuff here...

iUserLevel := E_User_Level.eUser_Level_none;

// main

stHmi.stOut.stCommon.stMain.stButton_Home.stName		:= stTextListGlobal.stText_Home;
stHmi.stOut.stCommon.stMain.stButton_Step.stName		:= stTextListGlobal.stText_Step;
stHmi.stOut.stCommon.stMain.stButton_Reset.stName		:= stTextListGlobal.stText_Reset;
stHmi.stOut.stCommon.stMain.stButton_CycleStop.stName	:= stTextListGlobal.stText_CycleStop;
stHmi.stOut.stCommon.stMain.stButton_Start.stName		:= stTextListGlobal.stText_Start;
stHmi.stOut.stCommon.stMain.stButton_Stop.stName		:= stTextListGlobal.stText_Stop;
stHmi.stOut.stCommon.stMain.stButton_PlantLight.stName	:= stTextListGlobal.stText_PlantLight;

// OP modes
stHmi.stOut.stCommon.stMain.stSwitch_OPM_1 := Const.stTextListGlobal.stText_off;
stHmi.stOut.stCommon.stMain.stSwitch_OPM_2 := Const.stTextListGlobal.stText_Manual;
stHmi.stOut.stCommon.stMain.stSwitch_OPM_3 := Const.stTextListGlobal.stText_Setup;
stHmi.stOut.stCommon.stMain.stSwitch_OPM_4 := Const.stTextListGlobal.stText_Auto;
	                                            
stHmi.stOut.stCommon.stMain.stButton_OPM_Auto.stName	:= stTextListGlobal.stText_OPM_Auto;
stHmi.stOut.stCommon.stMain.stButton_OPM_Step.stName	:= stTextListGlobal.stText_OPM_Step;
stHmi.stOut.stCommon.stMain.stButton_OPM_Manual.stName	:= stTextListGlobal.stText_OPM_Manual;

// user mgmt
stHmi.stOut.stCommon.stUserMgmt.stButton_LogOut.stName	:= stTextListGlobal.stText_logout;
stHmi.stOut.stCommon.stUserMgmt.stButton_LogIn.stName	:= stTextListGlobal.stText_login;
stHmi.stOut.stCommon.stUserMgmt.stButton_Submit.stName	:= stTextListGlobal.stText_submit;
//stHmi.stOut.stCommon.stUserManagment.stUserLevel		:= stUserLevel;

FOR ii := 1 TO E_Module.eModule_nMaxIdx - 1 DO
	stHmi.stOut.stCommon.arrStModule[ii].stButton_OPM_Auto.stName := stTextListGlobal.stText_Auto;
	stHmi.stOut.stCommon.arrStModule[ii].stButton_OPM_Step.stName := stTextListGlobal.stText_Step;
	stHmi.stOut.stCommon.arrStModule[ii].stButton_OPM_Manual.stName:= stTextListGlobal.stText_Manual;
	
	stHmi.stOut.stCommon.arrStModule[ii].stButton_Home.stName := stTextListGlobal.stText_Home;
	stHmi.stOut.stCommon.arrStModule[ii].stButton_Step.stName := stTextListGlobal.stText_Step;
	stHmi.stOut.stCommon.arrStModule[ii].stButton_Reset.stName := stTextListGlobal.stText_Reset;
	stHmi.stOut.stCommon.arrStModule[ii].stButton_CycleStop.stName := stTextListGlobal.stText_CycleStop;
	stHmi.stOut.stCommon.arrStModule[ii].stButton_Start.stName := stTextListGlobal.stText_Start;
	stHmi.stOut.stCommon.arrStModule[ii].stButton_Stop.stName := stTextListGlobal.stText_Stop;	
	
	//stHmi.stOut.stCommon.arrStModule[ii].stInfo1 := stTextListGlobal.stText_AllOk;
	//stHmi.stOut.stCommon.arrStModule[ii].stInfo2 := stTextListGlobal.stText_AllOk;	
END_FOR

FOR ii := 1 TO E_Station.eStation_nMaxIdx - 1 DO
	stHmi.stOut.stCommon.arrStStation[ii].stButton_OPM_Auto.stName := stTextListGlobal.stText_Auto;
	stHmi.stOut.stCommon.arrStStation[ii].stButton_OPM_Step.stName := stTextListGlobal.stText_Step;
	stHmi.stOut.stCommon.arrStStation[ii].stButton_OPM_Manual.stName:= stTextListGlobal.stText_Manual;
	
	stHmi.stOut.stCommon.arrStStation[ii].stButton_Home.stName := stTextListGlobal.stText_Home;
	stHmi.stOut.stCommon.arrStStation[ii].stButton_Step.stName := stTextListGlobal.stText_Step;
	stHmi.stOut.stCommon.arrStStation[ii].stButton_Reset.stName := stTextListGlobal.stText_Reset;
	stHmi.stOut.stCommon.arrStStation[ii].stButton_CycleStop.stName := stTextListGlobal.stText_CycleStop;
	stHmi.stOut.stCommon.arrStStation[ii].stButton_Start.stName := stTextListGlobal.stText_Start;
	stHmi.stOut.stCommon.arrStStation[ii].stButton_Stop.stName := stTextListGlobal.stText_Stop;	
	
	//stHmi.stOut.stCommon.arrStStation[ii].stInfo1 := stTextListGlobal.stText_AllOk;
	//stHmi.stOut.stCommon.arrStStation[ii].stInfo2 := stTextListGlobal.stText_AllOk;	
END_FOR

FOR ii := 0 TO E_User.eUser_nMaxIdx - 1 DO
	stUserLevel[ii].iUserLevelMax:=(E_User_Level.eUser_Level_nMaxIdx);
END_FOR

// call axis mgr to set ref
M_AxisManagement();


//aSClearText[EN] := 'HMI init done.';
M_Init := TRUE;
END_METHOD

METHOD PRIVATE M_OnControlRequest : BOOL
VAR_INPUT
	IProvider 	: ITF_HMI_PROVIDER;
	eRequest	: E_HMI_CONTROL_REQUEST;
END_VAR
VAR
	xx 			: INT;
END_VAR
IF IProvider = 0 THEN
	RETURN;
END_IF

// loop provider, reset request on oher provider
FOR xx := 0 TO E_HMI_PROVIDER.eHmiProvider_nMaxIdx DO
	IF aiHmiProvider[xx] = 0 OR aiHmiProvider[xx] = IProvider THEN
		CONTINUE;
	END_IF
	
	CASE eRequest OF
		E_HMI_CONTROL_REQUEST.Default:
			aiHmiProvider[xx].RequestManualControl := FALSE;
			
		E_HMI_CONTROL_REQUEST.RecipeMgmtRequest:
			aiHmiProvider[xx].RequestRecipeMgmt := FALSE;
			
		E_HMI_CONTROL_REQUEST.SettingMgmtRequest:
			aiHmiProvider[xx].RequestSettingMgmt := FALSE;

		E_HMI_CONTROL_REQUEST.UserMgmtRequest:
			aiHmiProvider[xx].RequestUserMgmt := FALSE;
	END_CASE
END_FOR
END_METHOD

METHOD PRIVATE M_PlcToHmi : BOOL
VAR
	IMd	: IModule;
	ISt	: IStation;
END_VAR
// add/update system infos
M_AddSystemInfo();

// map safety infos to HMI
stHmi.stOut.stCommon.stSafety.bSAFE_ES_Ok := IO.stSafetyIO.stIn.bSAFE_ES_Ok;
stHmi.stOut.stCommon.stSafety.bSAFE_AREA_Ok := IO.stSafetyIO.stIn.bSAFE_AREA_Ok;
//stHmi.stOut.stCommon.stSafety.bSAFE_CONFIRMDEVICE_OK := IO.stSafetyIO.stIn.bSAFE_CONFIRMDEVICE_OK;
stHmi.stOut.stCommon.stSafety.bLedResetSafety := SEL(P_Safety.ErrorAckRequest, FALSE, stPulse.bToggle500ms);
stHmi.stOut.stCommon.stSafety.bLedResetAreaST10 := SEL(P_Safety.SafetyAreaOk_ST10, stPulse.bToggle500ms, FALSE);
stHmi.stOut.stCommon.stSafety.bLedResetAreaST33 := SEL(NOT P_Safety.EmergencyStopOk OR P_Safety.SafetyAreaOk_ST20, stPulse.bToggle500ms, FALSE);

// OP mode manual
stHmi.stOut.stCommon.stMain.stButton_OPM_Manual.stColor.color := F_ColorToStringHexColor(STATICS.stColor.Theme);
IF FALSE THEN
	stHmi.stOut.stCommon.stMain.stButton_OPM_Manual.stColor.color := F_ColorToStringHexColor(STATICS.stColor.Orange);
ELSIF stGlobalModuleInfo.bStation_Any_Manual AND stPulse.bToggle1000ms THEN
	stHmi.stOut.stCommon.stMain.stButton_OPM_Manual.stColor.color := F_ColorToStringHexColor(STATICS.stColor.Orange);	
END_IF

// OP mode auto
stHmi.stOut.stCommon.stMain.stButton_OPM_Auto.stColor.color := F_ColorToStringHexColor(STATICS.stColor.Theme);
IF stGlobalModuleInfo.bStation_All_Auto THEN
	stHmi.stOut.stCommon.stMain.stButton_OPM_Auto.stColor.color := F_ColorToStringHexColor(STATICS.stColor.LimeGreen);
ELSIF FALSE AND stPulse.bToggle1000ms THEN
	stHmi.stOut.stCommon.stMain.stButton_OPM_Auto.stColor.color := F_ColorToStringHexColor(STATICS.stColor.LimeGreen);	
END_IF

// OP mode step
stHmi.stOut.stCommon.stMain.stButton_OPM_Step.stColor.color := F_ColorToStringHexColor(STATICS.stColor.Theme);
IF FALSE THEN
	stHmi.stOut.stCommon.stMain.stButton_OPM_Step.stColor.color := F_ColorToStringHexColor(STATICS.stColor.White);
ELSIF stGlobalModuleInfo.bStation_Any_Step AND stPulse.bToggle1000ms THEN
	stHmi.stOut.stCommon.stMain.stButton_OPM_Step.stColor.color := F_ColorToStringHexColor(STATICS.stColor.White);	
END_IF

// home
stHmi.stOut.stCommon.stMain.stButton_Home.bLed := FALSE;
stHmi.stOut.stCommon.stMain.stButton_Home.stColor.color := F_ColorToStringHexColor(STATICS.stColor.Theme);
IF stGlobalModuleInfo.bStation_All_InHome THEN
	stHmi.stOut.stCommon.stMain.stButton_Home.bLed := TRUE;
	stHmi.stOut.stCommon.stMain.stButton_Home.stColor.color := F_ColorToStringHexColor(STATICS.stColor.LightBlue);
ELSIF stGlobalModuleInfo.bStation_Any_Homing AND stPulse.bToggle1000ms THEN
	stHmi.stOut.stCommon.stMain.stButton_Home.bLed := TRUE;
	stHmi.stOut.stCommon.stMain.stButton_Home.stColor.color := F_ColorToStringHexColor(STATICS.stColor.LightBlue);	
END_IF

// step
stHmi.stOut.stCommon.stMain.stButton_Step.bLed := FALSE;
stHmi.stOut.stCommon.stMain.stButton_Step.stColor.color := F_ColorToStringHexColor(STATICS.stColor.Theme);
IF FALSE THEN
	stHmi.stOut.stCommon.stMain.stButton_Step.bLed := TRUE;
	stHmi.stOut.stCommon.stMain.stButton_Step.stColor.color := F_ColorToStringHexColor(STATICS.stColor.White);
ELSIF stGlobalModuleInfo.bStation_Any_Step AND stPulse.bToggle1000ms THEN
	stHmi.stOut.stCommon.stMain.stButton_Step.bLed := TRUE;
	stHmi.stOut.stCommon.stMain.stButton_Step.stColor.color := F_ColorToStringHexColor(STATICS.stColor.White);	
END_IF

// start
stHmi.stOut.stCommon.stMain.stButton_Start.bLed := FALSE;
stHmi.stOut.stCommon.stMain.stButton_Start.stColor.color := F_ColorToStringHexColor(STATICS.stColor.Theme);
IF stGlobalModuleInfo.bStation_All_Started THEN
	stHmi.stOut.stCommon.stMain.stButton_Start.bLed := TRUE;
	stHmi.stOut.stCommon.stMain.stButton_Start.stColor.color := F_ColorToStringHexColor(STATICS.stColor.LimeGreen);
ELSIF stGlobalModuleInfo.bStation_All_Auto AND stPulse.bToggle1000ms THEN
	stHmi.stOut.stCommon.stMain.stButton_Start.bLed := TRUE;
	stHmi.stOut.stCommon.stMain.stButton_Start.stColor.color := F_ColorToStringHexColor(STATICS.stColor.LimeGreen);	
END_IF

// cycle stop
stHmi.stOut.stCommon.stMain.stButton_CycleStop.stColor.color := F_ColorToStringHexColor(STATICS.stColor.Theme);
IF stGlobalModuleInfo.bStation_All_Stopped THEN
	stHmi.stOut.stCommon.stMain.stButton_CycleStop.stColor.color := F_ColorToStringHexColor(STATICS.stColor.Red);
ELSIF FALSE AND stPulse.bToggle1000ms THEN
	stHmi.stOut.stCommon.stMain.stButton_CycleStop.stColor.color := F_ColorToStringHexColor(STATICS.stColor.Red);	
END_IF

// stop
stHmi.stOut.stCommon.stMain.stButton_Stop.stColor.color := F_ColorToStringHexColor(STATICS.stColor.Theme);
IF stGlobalModuleInfo.bStation_All_Stopped THEN
	stHmi.stOut.stCommon.stMain.stButton_Stop.stColor.color := F_ColorToStringHexColor(STATICS.stColor.Red);
ELSIF FALSE AND stPulse.bToggle1000ms THEN
	stHmi.stOut.stCommon.stMain.stButton_Stop.stColor.color := F_ColorToStringHexColor(STATICS.stColor.Red);	
END_IF

//reset button
stHmi.stOut.stCommon.stMain.stButton_Reset.bLed := FALSE;
stHmi.stOut.stCommon.stMain.stButton_Reset.stColor.color := F_ColorToStringHexColor(STATICS.stColor.Theme);
IF (stGlobalModuleInfo.bStation_Any_Error OR P_Safety.bError) AND stPulse.bToggle1000ms THEN
	stHmi.stOut.stCommon.stMain.stButton_Reset.bLed := TRUE;
	stHmi.stOut.stCommon.stMain.stButton_Reset.stColor.color := F_ColorToStringHexColor(STATICS.stColor.Red);
END_IF

// plant light
stHmi.stOut.stCommon.stMain.stButton_PlantLight.stColor.color := F_ColorToStringHexColor(STATICS.stColor.Theme);
//IF IO.stControlCabinetIO.stOut.bAktor_Schuetz_Anlagenbeleuchtung THEN
	stHmi.stOut.stCommon.stMain.stButton_PlantLight.stColor.color := F_ColorToStringHexColor(STATICS.stColor.Yellow);
//END_IF

// plant traffic light
stHmi.stOut.stCommon.stTrafficLight.bLedGN := FALSE;							// green
IF stGlobalModuleInfo.bStation_All_Started THEN
	stHmi.stOut.stCommon.stTrafficLight.bLedGN := TRUE;
ELSIF stGlobalModuleInfo.bStation_All_Auto THEN
	stHmi.stOut.stCommon.stTrafficLight.bLedGN := stPulse.bToggle1000ms;	
END_IF

stHmi.stOut.stCommon.stTrafficLight.bLedGE := FALSE;							// yellow
IF (IEvent.WarningActive <> 0) THEN
	stHmi.stOut.stCommon.stTrafficLight.bLedGE := TRUE;
ELSIF FALSE THEN
	stHmi.stOut.stCommon.stTrafficLight.bLedGE := stPulse.bToggle1000ms;	
END_IF

stHmi.stOut.stCommon.stTrafficLight.bLedRT := FALSE;							// red
IF (IEvent.ErrorActive <> 0) THEN
	stHmi.stOut.stCommon.stTrafficLight.bLedRT := TRUE;
ELSIF FALSE THEN
	stHmi.stOut.stCommon.stTrafficLight.bLedRT := stPulse.bToggle1000ms;	
END_IF

stHmi.stOut.stCommon.stTrafficLight.bLedBL := FALSE;							// blue
IF (IEvent.InfoActive <> 0) THEN
	stHmi.stOut.stCommon.stTrafficLight.bLedBL := TRUE;
ELSIF FALSE THEN
	stHmi.stOut.stCommon.stTrafficLight.bLedBL := stPulse.bToggle1000ms;	
END_IF

// settings
sChanges := sEmpty;
Services.bSettingsSaved := FALSE;
stHmi.stOut.stCommon.stSettings.stControlSetting_Plant.stButtonSave.stName := stTextListGlobal.stText_Save;
stHmi.stOut.stCommon.stSettings.stControlSetting_Product.stButtonSave.stName := stTextListGlobal.stText_Save;
stHmi.stOut.stCommon.stSettings.stControlSetting_Production.stButtonSave.stName := stTextListGlobal.stText_Save;
fbSettingsHandling(eUserLevel := HMI.eUserLevel, stControlSettingIn := stHmi.stIn.stSettings.stControlSetting_Plant, stControlSettingOut := stHmi.stOut.stCommon.stSettings.stControlSetting_Plant, stSettings := Services.stSettings.stPlant_Settings, stSettingsView := stHmi.stOut.stCommon.stSettings.stSettingViewPlant, sChanges := sChanges);
fbSettingsHandling(eUserLevel := HMI.eUserLevel, stControlSettingIn := stHmi.stIn.stSettings.stControlSetting_Product, stControlSettingOut := stHmi.stOut.stCommon.stSettings.stControlSetting_Product, stSettings := Services.stSettings.stProduct_Settings, stSettingsView := stHmi.stOut.stCommon.stSettings.stSettingViewProduct, sChanges := sChanges);
fbSettingsHandling(eUserLevel := HMI.eUserLevel, stControlSettingIn := stHmi.stIn.stSettings.stControlSetting_Production, stControlSettingOut := stHmi.stOut.stCommon.stSettings.stControlSetting_Production, stSettings := Services.stSettings.stProduction_Settings, stSettingsView := stHmi.stOut.stCommon.stSettings.stSettingViewProduction, sChanges := sChanges);

// modules, settings, nav buttons,.. out
FOR ii := 0 TO E_Module.eModule_nMaxIdx DO
	IF P_Plant.aIModule[ii] = 0 THEN
		CONTINUE;
	END_IF
	
	IMd := P_Plant.aIModule[ii];
	M_PlcToHmiModule(IMd);
END_FOR

// stations, settings, nav buttons,.. out
FOR ii := 0 TO E_Station.eStation_nMaxIdx DO
	IF P_Plant.aIStaton[ii] = 0 THEN
		CONTINUE;
	END_IF
	
	ISt := P_Plant.aIStaton[ii];
	M_PlcToHmiStation(ISt);
END_FOR

// map project specific out 
M_SpecificPlcOut();

// track settings changes
IF sChanges <> sEmpty THEN
	ILog.AddLog(Concat5('Settings Changed, ', 'EKS level: ', TO_STRING(HMI.eUserLevel), '. Changes: ', sChanges), 
				'HMI Controller', 
				E_LogLevel.eLogLevel_info);
END_IF
END_METHOD

METHOD PRIVATE M_PlcToHmiModule : BOOL
VAR_INPUT
	IMd				: IModule;
END_VAR
VAR
	xx				: INT;
	nModuleIndex	: INT;
END_VAR
// set up texts
nModuleIndex := IMd.Module;
stHmi.stOut.stCommon.arrStModule[nModuleIndex].stName := IMd.Name;
stHmi.stOut.stCommon.arrStModule[nModuleIndex].stButtonNavigation.stName := IMd.Name;
stHmi.stOut.stCommon.arrStModule[nModuleIndex].stState_Auto := IMd.TextAuto;
stHmi.stOut.stCommon.arrStModule[nModuleIndex].stState_Home := IMd.TextHome;
stHmi.stOut.stCommon.stSettings.astSettingModules[nModuleIndex].stControlSetting.stButtonSave.stName := stTextListGlobal.stText_Save;

FOR xx := 0 TO CONST.iMaxIdxLocalStepChain DO
	stHmi.stOut.stCommon.arrStModule[nModuleIndex].aStepChainName[xx] := IMd.GetStepChainTest(xx);
END_FOR

// module state
stHmi.stOut.stCommon.arrStModule[nModuleIndex].stState := CONST.stTextListGlobal.stText_None;
IF IMd.State = E_ComponentState.eComponentState_none THEN
	stHmi.stOut.stCommon.arrStModule[nModuleIndex].stState := CONST.stTextListGlobal.stText_None;
ELSIF IMd.State = E_ComponentState.eComponentState_error THEN
	stHmi.stOut.stCommon.arrStModule[nModuleIndex].stState := CONST.stTextListGlobal.stText_Error;	
END_IF

// state OP mode buttons
stHmi.stOut.stCommon.arrStModule[nModuleIndex].stButton_OPM_Manual.stColor.color := F_ColorToStringHexColor(STATICS.stColor.Theme);
stHmi.stOut.stCommon.arrStModule[nModuleIndex].stButton_OPM_Auto.stColor.color := F_ColorToStringHexColor(STATICS.stColor.Theme);
stHmi.stOut.stCommon.arrStModule[nModuleIndex].stButton_OPM_Step.stColor.color := F_ColorToStringHexColor(STATICS.stColor.Theme);	
stHmi.stOut.stCommon.arrStModule[nModuleIndex].stButton_Reset.stColor.color := F_ColorToStringHexColor(STATICS.stColor.Theme);
stHmi.stOut.stCommon.arrStModule[nModuleIndex].stButton_Home.stColor.color := F_ColorToStringHexColor(STATICS.stColor.Theme);
stHmi.stOut.stCommon.arrStModule[nModuleIndex].stButton_Start.stColor.color := F_ColorToStringHexColor(STATICS.stColor.Theme);
stHmi.stOut.stCommon.arrStModule[nModuleIndex].stButton_CycleStop.stColor.color := F_ColorToStringHexColor(STATICS.stColor.Theme);
stHmi.stOut.stCommon.arrStModule[nModuleIndex].stButton_Stop.stColor.color := F_ColorToStringHexColor(STATICS.stColor.Theme);
stHmi.stOut.stCommon.arrStModule[nModuleIndex].stButton_Reset.stColor.color := F_ColorToStringHexColor(STATICS.stColor.Theme);

// op modes
stHmi.stOut.stCommon.arrStModule[nModuleIndex].stManual.bManualMode := IMd.OpMode = E_OpMode.eOpMode_manual;
IF IMd.OpMode = E_OpMode.eOpMode_manual THEN
	stHmi.stOut.stCommon.arrStModule[nModuleIndex].stButton_OPM_Manual.stColor.color := F_ColorToStringHexColor(STATICS.stColor.Orange);
	stHmi.stOut.stCommon.arrStModule[nModuleIndex].stButtonNavigation.stColor := stHmi.stOut.stCommon.arrStModule[nModuleIndex].stButton_OPM_Manual.stColor;
END_IF
IF IMd.OpMode = E_OpMode.eOpMode_auto THEN
	stHmi.stOut.stCommon.arrStModule[nModuleIndex].stButton_OPM_Auto.stColor.color := F_ColorToStringHexColor(STATICS.stColor.LimeGreen);
	stHmi.stOut.stCommon.arrStModule[nModuleIndex].stButtonNavigation.stColor := stHmi.stOut.stCommon.arrStModule[nModuleIndex].stButton_OPM_Auto.stColor;
END_IF
IF IMd.OpMode = E_OpMode.eOpMode_step THEN
	stHmi.stOut.stCommon.arrStModule[nModuleIndex].stButton_OPM_Step.stColor.color := F_ColorToStringHexColor(STATICS.stColor.White);
	stHmi.stOut.stCommon.arrStModule[nModuleIndex].stButtonNavigation.stColor.color := SEL(stPulse.bToggle1000ms OR IMd.RunCycle, F_ColorToStringHexColor(STATICS.stColor.Theme), stHmi.stOut.stCommon.arrStModule[nModuleIndex].stButton_OPM_Step.stColor.color);
END_IF

// state button home
IF IMd.InHome THEN
	stHmi.stOut.stCommon.arrStModule[nModuleIndex].stButton_Home.stColor.color := F_ColorToStringHexColor(STATICS.stColor.LightBlue);
	stHmi.stOut.stCommon.arrStModule[nModuleIndex].stButtonNavigation.stColor := stHmi.stOut.stCommon.arrStModule[nModuleIndex].stButton_Home.stColor;
END_IF

// state button start
IF ((IMd.OpMode = E_OpMode.eOpMode_auto OR IMd.OpMode = E_OpMode.eOpMode_step) AND IMd.RunCycle) THEN
	stHmi.stOut.stCommon.arrStModule[nModuleIndex].stButton_Start.stColor.color := F_ColorToStringHexColor(STATICS.stColor.LimeGreen);
ELSIF (IMd.OpMode = E_OpMode.eOpMode_step) THEN
	stHmi.stOut.stCommon.arrStModule[nModuleIndex].stButton_Start.stColor.color := F_ColorToStringHexColor(STATICS.stColor.White);
END_IF

// state button stop/cycle stop
IF IMd.Stopped THEN
	stHmi.stOut.stCommon.arrStModule[nModuleIndex].stButton_Stop.stColor.color := F_ColorToStringHexColor(STATICS.stColor.Red);
	stHmi.stOut.stCommon.arrStModule[nModuleIndex].stButton_CycleStop.stColor.color := F_ColorToStringHexColor(STATICS.stColor.Red);	
END_IF

// state button reset
IF IMd.State = E_ComponentState.eComponentState_error AND stPulse.bToggle1000ms THEN
	stHmi.stOut.stCommon.arrStModule[nModuleIndex].stButton_Reset.stColor.color := F_ColorToStringHexColor(STATICS.stColor.Red);
	stHmi.stOut.stCommon.arrStModule[nModuleIndex].stButtonNavigation.stColor := stHmi.stOut.stCommon.arrStModule[nModuleIndex].stButton_Reset.stColor;
END_IF

// module monitoring
fbMonitoringHandling(nDigits := 3, 
						stMonitoring := stHmi.stOut.stCommon.stMonitoring.astMonitoringModule[nModuleIndex].astMonitoring, 
						stMonitoringView := stHmi.stOut.stCommon.stMonitoring.astMonitoringModule[nModuleIndex].astMonitoringView);

// module settings
fbSettingsHandling(eUserLevel := HMI.eUserLevel, 
						stControlSettingIn := stHmi.stIn.stSettings.astControlSetting_Modules[nModuleIndex], 
						stControlSettingOut := stHmi.stOut.stCommon.stSettings.astSettingModules[nModuleIndex].stControlSetting, 
						stSettings := Services.stSettings.stModuleSettings[nModuleIndex].stDynStationSettings,
						stSettingsView := stHmi.stOut.stCommon.stSettings.astSettingModules[nModuleIndex].stSettingView,
					sChanges := sChanges);
END_METHOD

METHOD PRIVATE M_PlcToHmiStation : BOOL
VAR_INPUT
	ISt				: IStation;
END_VAR
VAR
	xx				: INT;
	nStationIndex	: INT;
END_VAR
// set up texts
nStationIndex := Ist.Station;
stHmi.stOut.stCommon.arrStStation[nStationIndex].stName := ISt.Name;
stHmi.stOut.stCommon.arrStStation[nStationIndex].stButtonNavigation.stName := ISt.Name;
stHmi.stOut.stCommon.arrStStation[nStationIndex].stState_Auto := ISt.TextAuto;
stHmi.stOut.stCommon.arrStStation[nStationIndex].stState_Home := ISt.TextHome;
stHmi.stOut.stCommon.stSettings.astSettingStations[nStationIndex].stControlSetting.stButtonSave.stName := stTextListGlobal.stText_Save;

FOR xx := 0 TO CONST.iMaxIdxLocalStepChain DO
	stHmi.stOut.stCommon.arrStStation[nStationIndex].aStepChainName[xx] := ISt.GetStepChainTest(xx);
END_FOR

// station state
stHmi.stOut.stCommon.arrStStation[nStationIndex].stState_Station := CONST.stTextListGlobal.stText_None;
IF Ist.State = E_ComponentState.eComponentState_none THEN
	stHmi.stOut.stCommon.arrStStation[nStationIndex].stState_Station := CONST.stTextListGlobal.stText_None;
ELSIF Ist.State = E_ComponentState.eComponentState_error THEN
	stHmi.stOut.stCommon.arrStStation[nStationIndex].stState_Station := CONST.stTextListGlobal.stText_Error;	
END_IF

// state OP mode buttons
stHmi.stOut.stCommon.arrStStation[nStationIndex].stButton_OPM_Manual.stColor.color := F_ColorToStringHexColor(STATICS.stColor.Theme);
stHmi.stOut.stCommon.arrStStation[nStationIndex].stButton_OPM_Auto.stColor.color := F_ColorToStringHexColor(STATICS.stColor.Theme);
stHmi.stOut.stCommon.arrStStation[nStationIndex].stButton_OPM_Step.stColor.color := F_ColorToStringHexColor(STATICS.stColor.Theme);	
stHmi.stOut.stCommon.arrStStation[nStationIndex].stButton_Reset.stColor.color := F_ColorToStringHexColor(STATICS.stColor.Theme);
stHmi.stOut.stCommon.arrStStation[nStationIndex].stButton_Home.stColor.color := F_ColorToStringHexColor(STATICS.stColor.Theme);
stHmi.stOut.stCommon.arrStStation[nStationIndex].stButton_Start.stColor.color := F_ColorToStringHexColor(STATICS.stColor.Theme);
stHmi.stOut.stCommon.arrStStation[nStationIndex].stButton_CycleStop.stColor.color := F_ColorToStringHexColor(STATICS.stColor.Theme);
stHmi.stOut.stCommon.arrStStation[nStationIndex].stButton_Stop.stColor.color := F_ColorToStringHexColor(STATICS.stColor.Theme);
stHmi.stOut.stCommon.arrStStation[nStationIndex].stButton_Reset.stColor.color := F_ColorToStringHexColor(STATICS.stColor.Theme);

// op modes
stHmi.stOut.stCommon.arrStStation[nStationIndex].stManual.bManualMode := Ist.OpMode = E_OpMode.eOpMode_manual;
IF Ist.OpMode = E_OpMode.eOpMode_manual THEN
	stHmi.stOut.stCommon.arrStStation[nStationIndex].stButton_OPM_Manual.stColor.color := F_ColorToStringHexColor(STATICS.stColor.Orange);
	stHmi.stOut.stCommon.arrStStation[nStationIndex].stButtonNavigation.stColor := stHmi.stOut.stCommon.arrStStation[nStationIndex].stButton_OPM_Manual.stColor;
END_IF
IF Ist.OpMode = E_OpMode.eOpMode_auto THEN
	stHmi.stOut.stCommon.arrStStation[nStationIndex].stButton_OPM_Auto.stColor.color := F_ColorToStringHexColor(STATICS.stColor.LimeGreen);
	stHmi.stOut.stCommon.arrStStation[nStationIndex].stButtonNavigation.stColor := stHmi.stOut.stCommon.arrStStation[nStationIndex].stButton_OPM_Auto.stColor;
END_IF
IF Ist.OpMode = E_OpMode.eOpMode_step THEN
	stHmi.stOut.stCommon.arrStStation[nStationIndex].stButton_OPM_Step.stColor.color := F_ColorToStringHexColor(STATICS.stColor.White);
	stHmi.stOut.stCommon.arrStStation[nStationIndex].stButtonNavigation.stColor.color := SEL(stPulse.bToggle1000ms OR Ist.RunCycle, F_ColorToStringHexColor(STATICS.stColor.Theme), stHmi.stOut.stCommon.arrStStation[nStationIndex].stButton_OPM_Step.stColor.color);
END_IF

// state button home
IF Ist.InHome THEN
	stHmi.stOut.stCommon.arrStStation[nStationIndex].stButton_Home.stColor.color := F_ColorToStringHexColor(STATICS.stColor.LightBlue);
	stHmi.stOut.stCommon.arrStStation[nStationIndex].stButtonNavigation.stColor := stHmi.stOut.stCommon.arrStStation[nStationIndex].stButton_Home.stColor;
END_IF

// state button start
IF ((Ist.OpMode = E_OpMode.eOpMode_auto OR Ist.OpMode = E_OpMode.eOpMode_step) AND Ist.RunCycle) THEN
	stHmi.stOut.stCommon.arrStStation[nStationIndex].stButton_Start.stColor.color := F_ColorToStringHexColor(STATICS.stColor.LimeGreen);
ELSIF (Ist.OpMode = E_OpMode.eOpMode_step) THEN
	stHmi.stOut.stCommon.arrStStation[nStationIndex].stButton_Start.stColor.color := F_ColorToStringHexColor(STATICS.stColor.White);
END_IF

// state button stop/cycle stop
IF Ist.Stopped THEN
	stHmi.stOut.stCommon.arrStStation[nStationIndex].stButton_Stop.stColor.color := F_ColorToStringHexColor(STATICS.stColor.Red);
	stHmi.stOut.stCommon.arrStStation[nStationIndex].stButton_CycleStop.stColor.color := F_ColorToStringHexColor(STATICS.stColor.Red);	
END_IF

// state button reset
IF Ist.State = E_ComponentState.eComponentState_error AND stPulse.bToggle1000ms THEN
	stHmi.stOut.stCommon.arrStStation[nStationIndex].stButton_Reset.stColor.color := F_ColorToStringHexColor(STATICS.stColor.Red);
	stHmi.stOut.stCommon.arrStStation[nStationIndex].stButtonNavigation.stColor := stHmi.stOut.stCommon.arrStStation[nStationIndex].stButton_Reset.stColor;
END_IF

// station monitoring
fbMonitoringHandling(nDigits := 3, 
						stMonitoring := stHmi.stOut.stCommon.stMonitoring.astMonitoringStation[nStationIndex].astMonitoring, 
						stMonitoringView := stHmi.stOut.stCommon.stMonitoring.astMonitoringStation[nStationIndex].astMonitoringView);

// station settings
fbSettingsHandling(eUserLevel := HMI.eUserLevel, 
						stControlSettingIn := stHmi.stIn.stSettings.astControlSetting_Stations[nStationIndex], 
						stControlSettingOut := stHmi.stOut.stCommon.stSettings.astSettingStations[nStationIndex].stControlSetting, 
						stSettings := Services.stSettings.stStationSettings[nStationIndex].stDynStationSettings,
						stSettingsView := stHmi.stOut.stCommon.stSettings.astSettingStations[nStationIndex].stSettingView,
					sChanges := sChanges);
END_METHOD

METHOD PRIVATE M_PlcToProvider : BOOL
VAR_IN_OUT
	IPrv		: ITF_HMI_PROVIDER;
END_VAR
VAR
	iMd, iSt 	: INT;
	stHmiOutPr 	: REFERENCE TO ST_HMI_OUT;
END_VAR
// main
stHmiOutPr REF= IPrv.ItfHmiOut;

//(mapping of common out not needed anymore, due to reference type!)
//stHmiOutPr.stCommon.stMain := stHmi.stOut.stCommon.stMain;
//	 
//// modules, just map
//FOR iMd := 0 TO E_Module.eModule_nMaxIdx DO
//	IF P_Plant.aIModule[iMd] = 0 THEN
//		CONTINUE;
//	END_IF
//	stHmiOutPr.arrStModule[iMd] := stHmi.stOut.arrStModule[iMd]; 
//END_FOR
//	 
//// stations, just map
//FOR iSt := 0 TO E_Station.eStation_nMaxIdx DO
//	IF P_Plant.aIStaton[iSt] = 0 THEN
//		CONTINUE;
//	END_IF
//	stHmiOutPr.arrStStation[iSt] := stHmi.stOut.arrStStation[iSt]; 
//END_FOR
//
//// recipe, settings, safety, user mgmt, traffic LEDs and system info
//stHmiOutPr.stRecipe := stHmi.stOut.stRecipe;
//stHmiOutPr.stSettings := stHmi.stOut.stSettings;
//stHmiOutPr.stMonitoring := stHmi.stOut.stMonitoring;
//stHmiOutPr.stSafety := stHmi.stOut.stSafety;
//stHmiOutPr.stUserMgmt := stHmi.stOut.stUserMgmt;
//stHmiOutPr.stTrafficLight := stHmi.stOut.stTrafficLight;
//stHmiOutPr.aSystemInfos := stHmi.stOut.aSystemInfos;
	 
// additional, project specific
M_SpecificProviderOut(stHmiOutPr);
END_METHOD

METHOD PRIVATE M_ProviderToPlc : BOOL
VAR_IN_OUT
	IPrv		: ITF_HMI_PROVIDER;
	fbPrvRqTrig	: FB_ProviderRequestTrigger;
END_VAR
VAR
	iMd, iSt 	: INT;
	stHmiInPr 	: REFERENCE TO ST_HMI_IN;
END_VAR
// main
stHmiInPr REF= IPrv.ItfHmiIn;
M_CombineCommonSignals(stHmi.stIn.stMain, stHmiInPr.stMain);
	 
// modules
FOR iMd := 0 TO E_Module.eModule_nMaxIdx DO
	IF P_Plant.aIModule[iMd] = 0 THEN
		CONTINUE;
	END_IF
	M_CombineCommonSignals(stHmi.stIn.arrStModule[iMd], stHmiInPr.arrStModule[iMd]);
	F_OR_REF(stHmi.stIn.arrStModule[iMd].stButtonNavigation.bClick, stHmiInPr.arrStModule[iMd].stButtonNavigation.bClick);
	
	IF IPrv.RequestManualControl THEN
		stHmi.stIn.arrStModule[iMd].iStepchain := stHmiInPr.arrStModule[iMd].iStepchain;
		stHmi.stIn.arrStModule[iMd].stManual := stHmiInPr.arrStModule[iMd].stManual;
	END_IF
END_FOR

// stations
FOR iSt := 0 TO E_Station.eStation_nMaxIdx DO
	IF P_Plant.aIStaton[iSt] = 0 THEN
		CONTINUE;
	END_IF
	M_CombineCommonSignals(stHmi.stIn.arrStStation[iSt], stHmiInPr.arrStStation[iSt]);
	F_OR_REF(stHmi.stIn.arrStStation[iSt].stButtonNavigation.bClick, stHmiInPr.arrStStation[iSt].stButtonNavigation.bClick);
	
	IF IPrv.RequestManualControl THEN
		stHmi.stIn.arrStStation[iSt].iStepchain := stHmiInPr.arrStStation[iSt].iStepchain;
		stHmi.stIn.arrStStation[iSt].stManual := stHmiInPr.arrStStation[iSt].stManual;
	END_IF
END_FOR

// recipe
IF IPrv.RequestRecipeMgmt THEN
	stHmi.stIn.stRecipe := stHmiInPr.stRecipe;
END_IF
	 
// settings
IF IPrv.RequestSettingMgmt THEN
	stHmi.stIn.stSettings := stHmiInPr.stSettings;
END_IF

// special
F_OR_REF(stHmi.stIn.stSpecial.stButton_LedTest.bClick, stHmiInPr.stSpecial.stButton_LedTest.bClick);
F_OR_REF(stHmi.stIn.stSpecial.stButton_CloseHmi.bClick, stHmiInPr.stSpecial.stButton_CloseHmi.bClick);
F_OR_REF(stHmi.stIn.stSpecial.stButton_SetSystemTime.bClick, stHmiInPr.stSpecial.stButton_SetSystemTime.bClick);
F_OR_REF(stHmi.stIn.stSpecial.stButton_Eplan.bClick, stHmiInPr.stSpecial.stButton_Eplan.bClick);
F_OR_REF(stHmi.stIn.stSpecial.stButton_Calculator.bClick, stHmiInPr.stSpecial.stButton_Calculator.bClick);
F_OR_REF(stHmi.stIn.stSpecial.stButton_KeyenceAutoIdNetwNav.bClick, stHmiInPr.stSpecial.stButton_KeyenceAutoIdNetwNav.bClick);
F_OR_REF(stHmi.stIn.stSpecial.stButton_KeyenceIv2Nav.bClick, stHmiInPr.stSpecial.stButton_KeyenceIv2Nav.bClick);
F_OR_REF(stHmi.stIn.stSpecial.stButton_CleanScreen.bClick, stHmiInPr.stSpecial.stButton_CleanScreen.bClick);

// user mgmt
IF IPrv.RequestRecipeMgmt THEN
	stHmi.stIn.stUserMgmt := stHmiInPr.stUserMgmt;
END_IF

// additional, project specific
M_SpecificProviderIn(IPrv, stHmiInPr);

// auto handle control request (Bedienhoheit)
fbPrvRqTrig(IProvider := IPrv);
IF fbPrvRqTrig.bManCtrlReq THEN
	M_OnControlRequest(IProvider := IPrv, E_HMI_CONTROL_REQUEST.Default);
ELSIF fbPrvRqTrig.bRecipeMgmtRequest THEN
	M_OnControlRequest(IProvider := IPrv, E_HMI_CONTROL_REQUEST.RecipeMgmtRequest);
ELSIF fbPrvRqTrig.bSettingMgmtRequest THEN
	M_OnControlRequest(IProvider := IPrv, E_HMI_CONTROL_REQUEST.SettingMgmtRequest);
ELSIF fbPrvRqTrig.bUserMgmtRequest THEN
	M_OnControlRequest(IProvider := IPrv, E_HMI_CONTROL_REQUEST.UserMgmtRequest);
END_IF
END_METHOD

METHOD INTERNAL M_RegisterProvider : BOOL
VAR_INPUT
	IProvider : ITF_HMI_PROVIDER;
END_VAR
aiHmiProvider[IProvider.Provider] := IProvider;
END_METHOD

/// resets all notification flags and reset-needed state 
METHOD M_Reset
VAR
	iPr : INT;
END_VAR

// RESET
IEvent.Reset();

FOR ii := 0 TO E_HMI_PROVIDER.eHmiProvider_nMaxIdx DO
	IF aiHmiProvider[iPr] = 0 THEN
		CONTINUE;
	END_IF
	
	aiHmiProvider[iPr].M_Reset();
END_FOR

// reset LED test
stHmi.stIn.stSpecial.stButton_LedTest.bClick := FALSE;
END_METHOD

METHOD M_SetReferences : BOOL
VAR_IN_OUT
	IEventHndler : FB_EventHandler;
END_VAR
HMI.stHmi.stOut.stCommon REF= stHmiBaseOut;
IEvent := IEventHndler;
M_SetReferences := TRUE;
END_METHOD

METHOD PRIVATE M_SpecificPlcOut : BOOL
VAR
END_VAR
// additional, project specific OUT (safety)

// opn door
//stHmi.stOut.stButtonDoorOpen.bLed := FALSE;
//IF NOT P_Safety.SafetyArea1Ok THEN
//	stHmi.stOut.stButtonDoorOpen.bLed := TRUE;
//ELSIF (NOT P_Safety.SafetyArea1Ok) AND stPulse.bToggle1000ms THEN
//	stHmi.stOut.stButtonDoorOpen.bLed := TRUE;	
//END_IF
//
//// cls door
//stHmi.stOut.stButtonDoorClose.bLed := FALSE;
//IF  P_Safety.SafetyArea1Ok THEN
//	stHmi.stOut.stButtonDoorClose.bLed := TRUE;
//ELSIF (NOT P_Safety.SafetyArea1Ok ) AND stPulse.bToggle1000ms 
//	AND NOT (NOT P_Safety.SafetyArea1Ok )
//THEN
//	stHmi.stOut.stButtonDoorClose.bLed := TRUE;	
//END_IF

// confirm
//stHmi.stOut.stButtonConfirm.bLed := FALSE;
//IF stHmi.stIn.stSafety.bConfirm THEN
//	stHmi.stOut.stButtonConfirm.bLed := TRUE;
//END_IF

// station specific..

M_SpecificPlcOut := TRUE;
END_METHOD

METHOD PRIVATE M_SpecificProviderIn : BOOL
VAR_IN_OUT
	IPrv		: ITF_HMI_PROVIDER;
	stHmiInPr	: ST_HMI_IN;
END_VAR

VAR
	
	//stHmiInPr 	: REFERENCE TO ST_HMI_IN;
END_VAR

//stHmiInPr REF= IPrv.ItfHmiIn;

// additional, project specific IN
F_OR_REF(stHmi.stIn.stSafety.bQuitSafety, stHmiInPr.stSafety.bQuitSafety);
F_OR_REF(stHmi.stIn.stSafety.bQuitAreaST10, stHmiInPr.stSafety.bQuitAreaST10);
F_OR_REF(stHmi.stIn.stSafety.bUnlockDoorST33, stHmiInPr.stSafety.bUnlockDoorST33);

F_OR_REF(stHmi.stIn.arrStModule[E_Module.eModule_M001].stButton_Reset.bClick, stHmiInPr.stM001.bQuit);

F_OR_REF(stHmi.stIn.stSt010.bJogCh1Inside, stHmiInPr.stSt010.bJogCh1Inside);
F_OR_REF(stHmi.stIn.stSt010.bJogCh2Inside, stHmiInPr.stSt010.bJogCh2Inside);
F_OR_REF(stHmi.stIn.stSt010.bJogCh1Ouside, stHmiInPr.stSt010.bJogCh1Ouside);
F_OR_REF(stHmi.stIn.stSt010.bJogCh2Ouside, stHmiInPr.stSt010.bJogCh2Ouside);
F_OR_REF(stHmi.stIn.stSt010.bJogDown, stHmiInPr.stSt010.bJogDown);
F_OR_REF(stHmi.stIn.stSt010.bJogUp, stHmiInPr.stSt010.bJogUp);
F_OR_REF(stHmi.stIn.stSt010.bSpeed, stHmiInPr.stSt010.bSpeed);
F_OR_REF(stHmi.stIn.stSt010.bJog, stHmiInPr.stSt010.bJog);

F_OR_REF(stHmi.stIn.arrStStation[E_Station.eStation_ST010_OvenA].stButton_OPM_Manual.bClick, stHmiInPr.stSt010.bManual);
F_OR_REF(stHmi.stIn.arrStStation[E_Station.eStation_ST010_OvenA].stButton_Reset.bClick, stHmiInPr.stSt010.bQuit);

stHmiInPr.arrStStation[E_Station.eStation_ST010_OvenA].stManual.stManualAxis.eJogMode := stHmi.stIn.arrStStation[E_Station.eStation_ST010_OvenA].stManual.stManualAxis.eJogMode;
IF stHmiInPr.stSt010.bJog THEN

	IF 	stHmi.stIn.arrStStation[E_Station.eStation_ST010_OvenA].stManual.stManualAxis.eJogMode <> E_Axis_JogMode.eJogMode_0 THEN
		stHmi.stIn.arrStStation[E_Station.eStation_ST010_OvenA].stManual.stManualAxis.eJogMode := E_Axis_JogMode.eJogMode_0;
	ELSE
		stHmi.stIn.arrStStation[E_Station.eStation_ST010_OvenA].stManual.stManualAxis.eJogMode :=  SEL(stHmiInPr.stSt010.bSpeed, E_Axis_JogMode.eJogMode_1, E_Axis_JogMode.eJogMode_2);
	END_IF

END_IF
	
	
F_OR_REF(stHmi.stIn.stSt020.bJogCh1Inside, stHmiInPr.stSt020.bJogCh1Inside);
F_OR_REF(stHmi.stIn.stSt020.bJogCh2Inside, stHmiInPr.stSt020.bJogCh2Inside);
F_OR_REF(stHmi.stIn.stSt020.bJogCh1Ouside, stHmiInPr.stSt020.bJogCh1Ouside);
F_OR_REF(stHmi.stIn.stSt020.bJogCh2Ouside, stHmiInPr.stSt020.bJogCh2Ouside);
F_OR_REF(stHmi.stIn.stSt020.bJogDown, stHmiInPr.stSt020.bJogDown);
F_OR_REF(stHmi.stIn.stSt020.bJogUp, stHmiInPr.stSt020.bJogUp);
F_OR_REF(stHmi.stIn.stSt020.bSpeed, stHmiInPr.stSt020.bSpeed);
F_OR_REF(stHmi.stIn.stSt020.bJog, stHmiInPr.stSt020.bJog);

F_OR_REF(stHmi.stIn.arrStStation[E_Station.eStation_ST020_OvenB].stButton_OPM_Manual.bClick, stHmiInPr.stSt020.bManual);
F_OR_REF(stHmi.stIn.arrStStation[E_Station.eStation_ST020_OvenB].stButton_Reset.bClick, stHmiInPr.stSt020.bQuit);


stHmiInPr.arrStStation[E_Station.eStation_ST020_OvenB].stManual.stManualAxis.eJogMode := stHmi.stIn.arrStStation[E_Station.eStation_ST020_OvenB].stManual.stManualAxis.eJogMode;
IF stHmiInPr.stSt020.bJog THEN

	IF 	stHmi.stIn.arrStStation[E_Station.eStation_ST020_OvenB].stManual.stManualAxis.eJogMode <> E_Axis_JogMode.eJogMode_0 THEN
		stHmi.stIn.arrStStation[E_Station.eStation_ST020_OvenB].stManual.stManualAxis.eJogMode := E_Axis_JogMode.eJogMode_0;
	ELSE
		stHmi.stIn.arrStStation[E_Station.eStation_ST020_OvenB].stManual.stManualAxis.eJogMode :=  SEL(stHmiInPr.stSt020.bSpeed, E_Axis_JogMode.eJogMode_1, E_Axis_JogMode.eJogMode_2);
	END_IF

END_IF


F_OR_REF(stHmi.stIn.stSt030.bJogXN, stHmiInPr.stSt030.bJogXN);
F_OR_REF(stHmi.stIn.stSt030.bJogXP, stHmiInPr.stSt030.bJogXP);
F_OR_REF(stHmi.stIn.stSt030.bJogYN, stHmiInPr.stSt030.bJogYN);
F_OR_REF(stHmi.stIn.stSt030.bJogYP, stHmiInPr.stSt030.bJogYP);
F_OR_REF(stHmi.stIn.stSt030.bJogZN, stHmiInPr.stSt030.bJogZN);
F_OR_REF(stHmi.stIn.stSt030.bJogZP, stHmiInPr.stSt030.bJogZP);
F_OR_REF(stHmi.stIn.stSt030.bSpeed, stHmiInPr.stSt030.bSpeed);
F_OR_REF(stHmi.stIn.stSt030.bJog, stHmiInPr.stSt030.bJog);

F_OR_REF(stHmi.stIn.arrStStation[E_Station.eStation_ST030_Handling].stButton_OPM_Manual.bClick, stHmiInPr.stSt030.bManual);
F_OR_REF(stHmi.stIn.arrStStation[E_Station.eStation_ST030_Handling].stButton_Reset.bClick, stHmiInPr.stSt030.bQuit);

stHmiInPr.arrStStation[E_Station.eStation_ST030_Handling].stManual.stManualAxis.eJogMode := stHmi.stIn.arrStStation[E_Station.eStation_ST030_Handling].stManual.stManualAxis.eJogMode;
IF stHmiInPr.stSt030.bJog THEN

	IF 	stHmi.stIn.arrStStation[E_Station.eStation_ST030_Handling].stManual.stManualAxis.eJogMode <> E_Axis_JogMode.eJogMode_0 THEN
		stHmi.stIn.arrStStation[E_Station.eStation_ST030_Handling].stManual.stManualAxis.eJogMode := E_Axis_JogMode.eJogMode_0;
	ELSE
		stHmi.stIn.arrStStation[E_Station.eStation_ST030_Handling].stManual.stManualAxis.eJogMode :=  SEL(stHmiInPr.stSt030.bSpeed, E_Axis_JogMode.eJogMode_1, E_Axis_JogMode.eJogMode_2);
	END_IF

END_IF

F_OR_REF(stHmi.stIn.stSt040.bJog01Down, stHmiInPr.stSt040.bJog01Down);
F_OR_REF(stHmi.stIn.stSt040.bJog01Up, stHmiInPr.stSt040.bJog01Up);
F_OR_REF(stHmi.stIn.stSt040.bJog02Down, stHmiInPr.stSt040.bJog02Down);
F_OR_REF(stHmi.stIn.stSt040.bJog02Up, stHmiInPr.stSt040.bJog02Up);
F_OR_REF(stHmi.stIn.stSt040.bSpeed, stHmiInPr.stSt010.bSpeed);
F_OR_REF(stHmi.stIn.stSt040.bJog, stHmiInPr.stSt010.bJog);

F_OR_REF(stHmi.stIn.stSt040.bJog, stHmiInPr.stSt040.bJog);F_OR_REF(stHmi.stIn.arrStStation[E_Station.eStation_ST040_Storage].stButton_OPM_Manual.bClick, stHmiInPr.stSt040.bManual);
F_OR_REF(stHmi.stIn.arrStStation[E_Station.eStation_ST040_Storage].stButton_Reset.bClick, stHmiInPr.stSt040.bQuit);

stHmiInPr.arrStStation[E_Station.eStation_ST040_Storage].stManual.stManualAxis.eJogMode := stHmi.stIn.arrStStation[E_Station.eStation_ST040_Storage].stManual.stManualAxis.eJogMode;
IF stHmiInPr.stSt040.bJog THEN

	IF 	stHmi.stIn.arrStStation[E_Station.eStation_ST040_Storage].stManual.stManualAxis.eJogMode <> E_Axis_JogMode.eJogMode_0 THEN
		stHmi.stIn.arrStStation[E_Station.eStation_ST040_Storage].stManual.stManualAxis.eJogMode := E_Axis_JogMode.eJogMode_0;
	ELSE
		stHmi.stIn.arrStStation[E_Station.eStation_ST040_Storage].stManual.stManualAxis.eJogMode :=  SEL(stHmiInPr.stSt040.bSpeed, E_Axis_JogMode.eJogMode_1, E_Axis_JogMode.eJogMode_2);
	END_IF

END_IF


// map override only from HW-provider (Poti)
IF IPrv.Provider = E_HMI_PROVIDER.eHmiProvider_HW THEN
	stHmi.stIn.iOverride := TO_INT(stHmiInPr.iOverride * 3.051851E-3);
END_IF

M_SpecificProviderIn := TRUE;
END_METHOD

METHOD PRIVATE M_SpecificProviderOut : BOOL
VAR_IN_OUT
	stHmiOutPr : ST_HMI_OUT;
END_VAR
// additional, project specific OUT to provider
stHmiOutPr.stM001 := stHmi.stOut.stM001;

stHmiOutPr.stSt010 := stHmi.stOut.stSt010;
stHmiOutPr.stSt020 := stHmi.stOut.stSt020;
stHmiOutPr.stSt030 := stHmi.stOut.stSt030;
stHmiOutPr.stSt040 := stHmi.stOut.stSt040;

M_SpecificProviderOut := TRUE;
END_METHOD

METHOD PRIVATE M_UpdateSystemInfo : BOOL
VAR_INPUT
	sName 	: STRING(31);
	sValue 	: STRING;
END_VAR
VAR_IN_OUT
	idx 	: INT;
END_VAR
IF idx < 0 OR idx > CONST.iMaxIdxSystemInfo THEN
	M_UpdateSystemInfo := FALSE;
	RETURN;
END_IF

stHmi.stOut.stCommon.aSystemInfos[idx].sName := sName;
stHmi.stOut.stCommon.aSystemInfos[idx].sValue := sValue;
idx := idx + 1;
M_UpdateSystemInfo := TRUE;
END_METHOD

METHOD M_UserManagement : INT
VAR_INPUT
END_VAR
tonUserLevelLogOut.IN:= (iUserLevel >= E_User_Level.eUser_Level_Maintenance);
tonUserLevelLogOut.PT:=T#15M;
tonUserLevelLogOut();

rTrigUserManagmentSubmit.CLK := stHmi.stIn.stUserMgmt.stButton_Submit.bClick;
rTrigUserManagmentSubmit();
rTrigUserManagmentLogIn.CLK := stHmi.stIn.stUserMgmt.stButton_LogIn.bClick;
rTrigUserManagmentLogIn();
rTrigUserManagmentLogOut.CLK := stHmi.stIn.stUserMgmt.stButton_LogOut.bClick;
rTrigUserManagmentLogOut();

IF rTrigUserManagmentLogIn.Q THEN
	IF (stHmi.stIn.stUserMgmt.sUserManagment_InputPassword = stUserLevel[stHmi.stIn.stUserMgmt.stControlObject.nSelectedRowIndex].sPassword) THEN
		stHmi.stIn.stUserMgmt.sUserManagment_InputPassword := '';
		//sPasswort := stHmi.stIn.stUserManagment.sUserManagment_InputPassword;
		iUserLevel := stUserLevel[stHmi.stIn.stUserMgmt.stControlObject.nSelectedRowIndex].iUserLevel;
		sUserLevelLastUser := stUserLevel[stHmi.stIn.stUserMgmt.stControlObject.nSelectedRowIndex].sName;
		sUserLevelLastUser := CONCAT(sUserLevelLastUser,'  Level: ');
		sUserLevelLastUser := CONCAT(sUserLevelLastUser,TO_STRING(iUserLevel));	
	ELSE
		;
	END_IF	
	//stHmi.stIn.stUserManagment.sUserManagment_InputPassword := '';
ELSIF tonUserLevelLogOut.Q OR rTrigUserManagmentLogOut.Q THEN
	iUserLevel := E_User_Level.eUser_Level_none;
	//stHmi.stIn.stUserManagment.sUserManagment_InputPassword := '';
END_IF

IF iIBN > 0 THEN
	iUserLevel := 6;
END_IF

IF tonUserLevelLogOut.Q THEN
	iUserLevel:= E_User_Level.eUser_Level_none;
END_IF

FOR ii:=0 TO (E_User_Level.eUser_Level_nMaxIdx-1) DO
	stHmi.stOut.stCommon.stUserMgmt.bUserLevel[ii]:=FALSE;
END_FOR

CASE iUserLevel OF

	E_User_Level.eUser_Level_none:
		stHmi.stOut.stCommon.stUserMgmt.sUserState:='Kein Benutzer';
		stHmi.stOut.stCommon.stUserMgmt.bUserLevel[0]:=TRUE;
		
	E_User_Level.eUser_Level_Operator:
		stHmi.stOut.stCommon.stUserMgmt.sUserState:=sUserLevelLastUser;
		stHmi.stOut.stCommon.stUserMgmt.bUserLevel[0]:=TRUE;		
		stHmi.stOut.stCommon.stUserMgmt.bUserLevel[1]:=TRUE;
		
	E_User_Level.eUser_Level_Manager:
		stHmi.stOut.stCommon.stUserMgmt.sUserState:=sUserLevelLastUser;
		stHmi.stOut.stCommon.stUserMgmt.bUserLevel[0]:=TRUE;		
		stHmi.stOut.stCommon.stUserMgmt.bUserLevel[1]:=TRUE;
		stHmi.stOut.stCommon.stUserMgmt.bUserLevel[2]:=TRUE;	
		
	E_User_Level.eUser_Level_Maintenance:
		stHmi.stOut.stCommon.stUserMgmt.sUserState:=sUserLevelLastUser;
		stHmi.stOut.stCommon.stUserMgmt.bUserLevel[0]:=TRUE;		
		stHmi.stOut.stCommon.stUserMgmt.bUserLevel[1]:=TRUE;
		stHmi.stOut.stCommon.stUserMgmt.bUserLevel[2]:=TRUE;		
		stHmi.stOut.stCommon.stUserMgmt.bUserLevel[3]:=TRUE;
		
	E_User_Level.eUser_Level_Level4:
		stHmi.stOut.stCommon.stUserMgmt.sUserState:=sUserLevelLastUser;
		stHmi.stOut.stCommon.stUserMgmt.bUserLevel[0]:=TRUE;		
		stHmi.stOut.stCommon.stUserMgmt.bUserLevel[1]:=TRUE;
		stHmi.stOut.stCommon.stUserMgmt.bUserLevel[2]:=TRUE;		
		stHmi.stOut.stCommon.stUserMgmt.bUserLevel[3]:=TRUE;
		stHmi.stOut.stCommon.stUserMgmt.bUserLevel[4]:=TRUE;		
	
	E_User_Level.eUser_Level_Admin:
		stHmi.stOut.stCommon.stUserMgmt.sUserState:=sUserLevelLastUser;
		stHmi.stOut.stCommon.stUserMgmt.bUserLevel[0]:=TRUE;		
		stHmi.stOut.stCommon.stUserMgmt.bUserLevel[1]:=TRUE;
		stHmi.stOut.stCommon.stUserMgmt.bUserLevel[2]:=TRUE;		
		stHmi.stOut.stCommon.stUserMgmt.bUserLevel[3]:=TRUE;
		stHmi.stOut.stCommon.stUserMgmt.bUserLevel[4]:=TRUE;		
		stHmi.stOut.stCommon.stUserMgmt.bUserLevel[5]:=TRUE;	
		
	E_User_Level.eUser_Level_Programmer:
		stHmi.stOut.stCommon.stUserMgmt.sUserState:=sUserLevelLastUser;
		stHmi.stOut.stCommon.stUserMgmt.bUserLevel[0]:=TRUE;		
		stHmi.stOut.stCommon.stUserMgmt.bUserLevel[1]:=TRUE;
		stHmi.stOut.stCommon.stUserMgmt.bUserLevel[2]:=TRUE;		
		stHmi.stOut.stCommon.stUserMgmt.bUserLevel[3]:=TRUE;
		stHmi.stOut.stCommon.stUserMgmt.bUserLevel[4]:=TRUE;		
		stHmi.stOut.stCommon.stUserMgmt.bUserLevel[5]:=TRUE;	
		stHmi.stOut.stCommon.stUserMgmt.bUserLevel[6]:=TRUE;			
ELSE
	stHmi.stOut.stCommon.stUserMgmt.sUserState:='Benutzer unbekannt';
END_CASE

iUserLevel:=LIMIT(0, iUserLevel, (E_User_Level.eUser_Level_nMaxIdx - 1));

stHmi.stOut.stCommon.stUserMgmt.bPasswordInputVisible := bPasswordSave;
stHmi.stOut.stCommon.stUserMgmt.bCreateDeleteUserVisible := iUserLevel >= E_User_Level.eUser_Level_Admin; // only Admin or programmer can delete a user


FOR ii:=0 TO (E_User.eUser_nMaxIdx-1) DO
	stHmi.stOut.stCommon.stUserMgmt.stUserLevel[ii].sName := stUserLevel[ii].sName;		
	stHmi.stOut.stCommon.stUserMgmt.stUserLevel[ii].iUserLevel := stUserLevel[ii].iUserLevel;
	stHmi.stOut.stCommon.stUserMgmt.stUserLevel[ii].iUserLevelMin := stUserLevel[ii].iUserLevelMin;
	stHmi.stOut.stCommon.stUserMgmt.stUserLevel[ii].iUserLevelMax := stUserLevel[ii].iUserLevelMax;
	IF (iUserLevel < E_User_Level.eUser_Level_Admin) AND (stUserLevel[ii].sName <> '')
	THEN
		stHmi.stOut.stCommon.stUserMgmt.stUserLevel[ii].sPassword:='*****';
	ELSIF (iUserLevel >= stUserLevel[ii].iUserLevel(* E_User_Level.eUser_Level_Admin*)) AND (stUserLevel[ii].sName <> '') THEN
		stHmi.stOut.stCommon.stUserMgmt.stUserLevel[ii].sPassword:=stUserLevel[ii].sPassword;
	ELSIF NOT (iUserLevel >= stUserLevel[ii].iUserLevel (*E_User_Level.eUser_Level_Admin*)) AND (stUserLevel[ii].sName <> '')  
	THEN
		stHmi.stOut.stCommon.stUserMgmt.stUserLevel[ii].sPassword:='*****';
	ELSE
		stHmi.stOut.stCommon.stUserMgmt.stUserLevel[ii].sPassword:='';
	END_IF
	IF (stHmi.stOut.stCommon.stUserMgmt.stUserLevel[ii].sName <> '') THEN
		CASE stHmi.stOut.stCommon.stUserMgmt.stUserLevel[ii].iUserLevel OF
			0:
				stHmi.stOut.stCommon.stUserMgmt.stUserLevel[ii].stUserLevelName := stTextListGlobal.stText_UserLevel_None;

			1:
				stHmi.stOut.stCommon.stUserMgmt.stUserLevel[ii].stUserLevelName := stTextListGlobal.stText_UserLevel_Operator;

			2:
				stHmi.stOut.stCommon.stUserMgmt.stUserLevel[ii].stUserLevelName := stTextListGlobal.stText_UserLevel_Manager;

			3:
				stHmi.stOut.stCommon.stUserMgmt.stUserLevel[ii].stUserLevelName := stTextListGlobal.stText_UserLevel_Maintenance;

			4:
				stHmi.stOut.stCommon.stUserMgmt.stUserLevel[ii].stUserLevelName := stTextListGlobal.stText_UserLevel_None;

			5:
				stHmi.stOut.stCommon.stUserMgmt.stUserLevel[ii].stUserLevelName := stTextListGlobal.stText_UserLevel_Admin;

			6:
				stHmi.stOut.stCommon.stUserMgmt.stUserLevel[ii].stUserLevelName := stTextListGlobal.stText_UserLevel_Programmer;		

		END_CASE
	END_IF
END_FOR

stHmi.stOut.stCommon.stUserMgmt.aUserLevelList[0] := stTextListGlobal.stText_UserLevel_None;
stHmi.stOut.stCommon.stUserMgmt.aUserLevelList[1] := stTextListGlobal.stText_UserLevel_Operator;
stHmi.stOut.stCommon.stUserMgmt.aUserLevelList[2] := stTextListGlobal.stText_UserLevel_Manager;
stHmi.stOut.stCommon.stUserMgmt.aUserLevelList[3] := stTextListGlobal.stText_UserLevel_Maintenance;
stHmi.stOut.stCommon.stUserMgmt.aUserLevelList[4] := stTextListGlobal.stText_UserLevel_None;
stHmi.stOut.stCommon.stUserMgmt.aUserLevelList[5] := stTextListGlobal.stText_UserLevel_Admin;
stHmi.stOut.stCommon.stUserMgmt.aUserLevelList[6] := stTextListGlobal.stText_UserLevel_Programmer;

IF fTrigUserManagmentSubmit.Q THEN
	stHmi.stIn.stUserMgmt.sUserManagment_InputString := '';
	stHmi.stIn.stUserMgmt.nUserManagment_InputUserLevel := 0;
END_IF

// Column of the grid
CASE stHmi.stIn.stUserMgmt.stControlObject.nSelectedColumIndex OF 
	// Name
	0:
		// selected col/row changed
		IF nUserManagemenetColumnIdx_Old <> stHmi.stIn.stUserMgmt.stControlObject.nSelectedColumIndex OR
		nUserManagemenetRowIdx_Old <> stHmi.stIn.stUserMgmt.stControlObject.nSelectedRowIndex THEN
			nUserManagemenetColumnIdx_Old := stHmi.stIn.stUserMgmt.stControlObject.nSelectedColumIndex;
			nUserManagemenetRowIdx_Old := stHmi.stIn.stUserMgmt.stControlObject.nSelectedRowIndex;
			stHmi.stIn.stUserMgmt.sUserManagment_InputString := stUserLevel[stHmi.stIn.stUserMgmt.stControlObject.nSelectedRowIndex].sName;
		END_IF
		stHmi.stOut.stCommon.stUserMgmt.stInputDisplayText := F_CreateDynText("Name", 0);
		stHmi.stOut.stCommon.stUserMgmt.bKeyboardInputVisible := stHmi.stOut.stCommon.stUserMgmt.bUserLevel[E_User_Level.eUser_Level_Admin] 
																	OR stHmi.stOut.stCommon.stUserMgmt.bUserLevel[E_User_Level.eUser_Level_Programmer];
		stHmi.stOut.stCommon.stUserMgmt.bNumpadInputVisible := FALSE;
		stHmi.stOut.stCommon.stUserMgmt.bUserLevelInputVisible := FALSE;
		//Reihe 1 - Name des Benutzers nur übernehmen wenn Admin
		IF stHmi.stOut.stCommon.stUserMgmt.bUserLevel[E_User_Level.eUser_Level_Admin] 
			OR stHmi.stOut.stCommon.stUserMgmt.bUserLevel[E_User_Level.eUser_Level_Programmer] 
		THEN
			IF rTrigUserManagmentSubmit.Q THEN
				IF ((iUserLevel = E_User_Level.eUser_Level_Admin)
					AND (stUserLevel[stHmi.stIn.stUserMgmt.stControlObject.nSelectedRowIndex].iUserLevel <= E_User_Level.eUser_Level_Admin))
					OR stHmi.stOut.stCommon.stUserMgmt.bUserLevel[E_User_Level.eUser_Level_Programmer]
				THEN	
					stUserLevel[stHmi.stIn.stUserMgmt.stControlObject.nSelectedRowIndex].sName := stHmi.stIn.stUserMgmt.sUserManagment_InputString;
				ELSE
					stHmi.stOut.stCommon.stUserMgmt.sUserState:='Benutzer level incorrect';
				END_IF
			END_IF
		END_IF

	// Passwort
	1:
		// selected col/row changed
		IF nUserManagemenetColumnIdx_Old <> stHmi.stIn.stUserMgmt.stControlObject.nSelectedColumIndex OR
		nUserManagemenetRowIdx_Old <> stHmi.stIn.stUserMgmt.stControlObject.nSelectedRowIndex THEN
			nUserManagemenetColumnIdx_Old := stHmi.stIn.stUserMgmt.stControlObject.nSelectedColumIndex;
			nUserManagemenetRowIdx_Old := stHmi.stIn.stUserMgmt.stControlObject.nSelectedRowIndex;
			stHmi.stIn.stUserMgmt.sUserManagment_InputString := '*****';
		END_IF
		stHmi.stOut.stCommon.stUserMgmt.stInputDisplayText := F_CreateDynText("Passwort", 0);
		stHmi.stOut.stCommon.stUserMgmt.bKeyboardInputVisible := stHmi.stOut.stCommon.stUserMgmt.bUserLevel[E_User_Level.eUser_Level_Admin] OR stHmi.stOut.stCommon.stUserMgmt.bUserLevel[E_User_Level.eUser_Level_Programmer];
		stHmi.stOut.stCommon.stUserMgmt.bNumpadInputVisible := FALSE;
		stHmi.stOut.stCommon.stUserMgmt.bUserLevelInputVisible := FALSE;
		//Reihe 2 - Passwort der Eingabe gleich hinterlegtem Passwort dann User aktivieren
		IF (stHmi.stOut.stCommon.stUserMgmt.bUserLevel[E_User_Level.eUser_Level_Admin] AND (stUserLevel[stHmi.stIn.stUserMgmt.stControlObject.nSelectedRowIndex].iUserLevel < E_User_Level.eUser_Level_Programmer)) 
			OR stHmi.stOut.stCommon.stUserMgmt.bUserLevel[E_User_Level.eUser_Level_Programmer] 
		THEN
			IF rTrigUserManagmentSubmit.Q  
				AND (stHmi.stIn.stUserMgmt.sUserManagment_InputString <> '') 
				AND (stHmi.stIn.stUserMgmt.sUserManagment_InputString <> '*****') THEN
				stUserLevel[stHmi.stIn.stUserMgmt.stControlObject.nSelectedRowIndex].sPassword := stHmi.stIn.stUserMgmt.sUserManagment_InputString;
			END_IF
		END_IF

	// Stufe
	2:
		// selected col/row changed
		IF nUserManagemenetColumnIdx_Old <> stHmi.stIn.stUserMgmt.stControlObject.nSelectedColumIndex OR
		nUserManagemenetRowIdx_Old <> stHmi.stIn.stUserMgmt.stControlObject.nSelectedRowIndex THEN
			nUserManagemenetColumnIdx_Old := stHmi.stIn.stUserMgmt.stControlObject.nSelectedColumIndex;
			nUserManagemenetRowIdx_Old := stHmi.stIn.stUserMgmt.stControlObject.nSelectedRowIndex;
			stHmi.stIn.stUserMgmt.nUserManagment_InputUserLevel := stUserLevel[stHmi.stIn.stUserMgmt.stControlObject.nSelectedRowIndex].iUserLevel;
		END_IF
		stHmi.stOut.stCommon.stUserMgmt.stInputDisplayText := F_CreateDynText("Stufe", 0);
		stHmi.stOut.stCommon.stUserMgmt.bKeyboardInputVisible := FALSE;
		stHmi.stOut.stCommon.stUserMgmt.bNumpadInputVisible := FALSE;
		stHmi.stOut.stCommon.stUserMgmt.bUserLevelInputVisible := stHmi.stOut.stCommon.stUserMgmt.bUserLevel[E_User_Level.eUser_Level_Admin];
		IF (stHmi.stOut.stCommon.stUserMgmt.bUserLevel[E_User_Level.eUser_Level_Admin] 
				AND (stUserLevel[stHmi.stIn.stUserMgmt.stControlObject.nSelectedRowIndex].iUserLevel < E_User_Level.eUser_Level_Programmer)
				AND (stHmi.stIn.stUserMgmt.nUserManagment_InputUserLevel < E_User_Level.eUser_Level_Programmer)) 
			OR stHmi.stOut.stCommon.stUserMgmt.bUserLevel[E_User_Level.eUser_Level_Programmer] 
		THEN
			IF rTrigUserManagmentSubmit.Q THEN
				stUserLevel[stHmi.stIn.stUserMgmt.stControlObject.nSelectedRowIndex].iUserLevel := stHmi.stIn.stUserMgmt.nUserManagment_InputUserLevel;
			END_IF
		END_IF

	ELSE
		//ELSE Alle Visible Rücksetzen
		stHmi.stOut.stCommon.stUserMgmt.bKeyboardInputVisible := FALSE;
		stHmi.stOut.stCommon.stUserMgmt.bNumpadInputVisible := FALSE;
		stHmi.stOut.stCommon.stUserMgmt.bUserLevelInputVisible := FALSE;
		
END_CASE

// Delete user
rTrigUserManagmentDelete( CLK := stHmi.stIn.stUserMgmt.bDeleteUser );
IF rTrigUserManagmentDelete.Q THEN
	IF ((iUserLevel >= E_User_Level.eUser_Level_Admin) AND (stUserLevel[stHmi.stIn.stUserMgmt.stControlObject.nSelectedRowIndex].iUserLevel < E_User_Level.eUser_Level_Programmer) ) 
		OR stHmi.stOut.stCommon.stUserMgmt.bUserLevel[E_User_Level.eUser_Level_Programmer]
	THEN
		stHmi.stOut.stCommon.stUserMgmt.stUserManagementMessage := F_CreateDynText("", 0);
		
		stUserLevel[stHmi.stIn.stUserMgmt.stControlObject.nSelectedRowIndex].sName  := '';
		stUserLevel[stHmi.stIn.stUserMgmt.stControlObject.nSelectedRowIndex].sPassword  := '';
		stUserLevel[stHmi.stIn.stUserMgmt.stControlObject.nSelectedRowIndex].iUserLevel := TO_INT( E_User_Level.eUser_Level_none );
		// message
		stHmi.stOut.stCommon.stUserMgmt.stUserManagementMessage := F_CreateDynText("Benutzer gelöscht!", 0);
	
	ELSIF stHmi.stIn.stUserMgmt.sCreateDeleteUserName = '' THEN
		stHmi.stOut.stCommon.stUserMgmt.stUserManagementMessage := F_CreateDynText("Benutzername ist leer!", 0);
	ELSIF stHmi.stIn.stUserMgmt.sCreateDeleteUserName <> stHmi.stIn.stUserMgmt.sCreateDeleteUserNameConfirm THEN
		stHmi.stOut.stCommon.stUserMgmt.stUserManagementMessage := F_CreateDynText("Benutzername bitte bestätigen!", 0);
	END_IF	
END_IF

HMI.eUserLevel := iUserLevel;
END_METHOD

END_PROGRAM

// ---- POUs/HMI/Utilities/FB_ProviderRequestTrigger.TcPOU
FUNCTION_BLOCK INTERNAL FB_ProviderRequestTrigger
VAR_INPUT
	IProvider 				: ITF_HMI_PROVIDER;
END_VAR
VAR_OUTPUT
	bManCtrlReq 			: BOOL;
	bRecipeMgmtRequest 		: BOOL;
	bSettingMgmtRequest 	: BOOL;
	bUserMgmtRequest 		: BOOL;
END_VAR
VAR
	fTrigManCtrlReq			: R_TRIG;
	fTrigRecipeMgmtReq		: R_TRIG;
	fTrigSettingsMgmtReq	: R_TRIG;
	fTrigUserMgmtReq		: R_TRIG;
END_VAR

IF (IProvider = 0) THEN
	RETURN;
END_IF

fTrigManCtrlReq(CLK := IProvider.RequestManualControl, Q => bManCtrlReq);
fTrigRecipeMgmtReq(CLK := IProvider.RequestRecipeMgmt, Q => bRecipeMgmtRequest);
fTrigSettingsMgmtReq(CLK := IProvider.RequestSettingMgmt, Q => bSettingMgmtRequest);
fTrigUserMgmtReq(CLK := IProvider.RequestUserMgmt, Q => bUserMgmtRequest);

END_FUNCTION_BLOCK

// ---- POUs/HMI/Utilities/FB_HmiBaseControlTrigger.TcPOU
FUNCTION_BLOCK INTERNAL FB_HmiBaseControlTrigger
VAR_INPUT
	stHmiToPlcIn 	: ST_DefaultHmiToPlc;
END_VAR
VAR_IN_OUT
	stHmiToPlcOut 	: ST_DefaultHmiToPlc;
END_VAR
VAR
	fTrigStart	: F_TRIG;
	fTrigStop	: F_TRIG;
	fTrigReset	: F_TRIG;
	fTrigTip	: F_TRIG;
	
	tonHome		: TON;
	rTrigHome	: R_TRIG;
	
	fTrigOpModeManual	: F_TRIG;
	fTrigOpModeAuto		: F_TRIG;
	fTrigOpModeStep		: F_TRIG;
END_VAR

fTrigStart(CLK := stHmiToPlcIn.bStart, Q => stHmiToPlcOut.bStart);
stHmiToPlcOut.bStop := stHmiToPlcIn.bStop;
stHmiToPlcOut.bFastStop := stHmiToPlcIn.bFastStop;
stHmiToPlcOut.eSafetyOpMode := stHmiToPlcIn.eSafetyOpMode;
fTrigReset(CLK := stHmiToPlcIn.bReset, Q => stHmiToPlcOut.bReset);
fTrigTip(CLK := stHmiToPlcIn.bStep, Q => stHmiToPlcOut.bStep);

tonHome(IN := stHmiToPlcIn.bHome, PT := T#1S);
rTrigHome(CLK := tonHome.Q, Q => stHmiToPlcOut.bHome);

fTrigOpModeManual(CLK := stHmiToPlcIn.bOpModeManual, Q => stHmiToPlcOut.bOpModeManual);
fTrigOpModeAuto(CLK := stHmiToPlcIn.bOpModeAuto, Q => stHmiToPlcOut.bOpModeAuto);
fTrigOpModeStep(CLK := stHmiToPlcIn.bOpModeStep, Q => stHmiToPlcOut.bOpModeStep);

END_FUNCTION_BLOCK

// ---- POUs/HMI/Utilities/SettingsHandling/FB_SettingsHandling.TcPOU
FUNCTION_BLOCK FB_SettingsHandling
VAR_INPUT
	eUserLevel			: E_User_Level;
END_VAR
VAR_IN_OUT
	stControlSettingIn	: ST_HMI_CONTROL_SETTING_ITEM_IN;
	stControlSettingOut	: ST_HMI_CONTROL_SETTING_ITEM_OUT;
	stSettings			: ARRAY[*] OF ST_Data_Item;
	stSettingsView		: ARRAY[*] OF ST_Data_Item_String;
	sChanges			: T_MaxString;
END_VAR
VAR
	ii, nLb, nUb	: DINT;
	rtSave			: R_TRIG;
	nColIndex,
	nRowIndex		: INT;
	tofInfo			: TOF;
	stInfo			: ST_Text;
END_VAR

nColIndex := TO_INT(stControlSettingIn.nSelectedColumIndex);
nRowIndex := TO_INT(stControlSettingIn.nSelectedRowIndex);

stControlSettingOut.stButtonSave.stColor.color := F_ColorToStringHexColor(STATICS.stColor.Theme);
IF stControlSettingIn.stButtonSave.bClick THEN
	stControlSettingOut.stButtonSave.stColor.color := F_ColorToStringHexColor(STATICS.stColor.LimeGreen);
END_IF

stControlSettingOut.bVisible_Bool := FALSE;
stControlSettingOut.bVisible_Float := FALSE;
stControlSettingOut.bVisible_Number := FALSE;
stControlSettingOut.bVisible_String := FALSE;
stControlSettingOut.bVisible_UserLevel := FALSE;
stControlSettingOut.bVisible_RecipeMode := FALSE;

stControlSettingOut.nUserLevelUsers := (E_User_Level.eUser_Level_nMaxIdx);
stControlSettingOut.aUserLevelUsers[E_User_Level.eUser_Level_none] := CONST.stTextListGlobal.stText_UserLevel00;
stControlSettingOut.aUserLevelUsers[E_User_Level.eUser_Level_Operator] := CONST.stTextListGlobal.stText_UserLevel01;
stControlSettingOut.aUserLevelUsers[E_User_Level.eUser_Level_Manager] := CONST.stTextListGlobal.stText_UserLevel02;
stControlSettingOut.aUserLevelUsers[E_User_Level.eUser_Level_Maintenance] := CONST.stTextListGlobal.stText_UserLevel03;
stControlSettingOut.aUserLevelUsers[E_User_Level.eUser_Level_Level4] := CONST.stTextListGlobal.stText_UserLevel04;
stControlSettingOut.aUserLevelUsers[E_User_Level.eUser_Level_Admin] := CONST.stTextListGlobal.stText_UserLevel05;
stControlSettingOut.aUserLevelUsers[E_User_Level.eUser_Level_Programmer] := CONST.stTextListGlobal.stText_UserLevel06;

stControlSettingOut.nRecipeMode := (E_RecipeMode.eRecipeMode_Max);
stControlSettingOut.aRecipeMode[E_RecipeMode.eRecipeMode_None] := CONST.stTextListGlobal.stText_Recipe_Mode_None;
stControlSettingOut.aRecipeMode[E_RecipeMode.eRecipeMode_ToFrom] := CONST.stTextListGlobal.stText_Recipe_Mode_ToFrom;

//clear settins view
nLb := LOWER_BOUND(stSettingsView, 1);
nUb := UPPER_BOUND(stSettingsView, 1);
FOR ii := nLb TO nUb DO
	MEMSET(ADR(stSettingsView[ii]),0,SIZEOF(stSettingsView[ii]));
END_FOR

nLb := MAX(nLb, LOWER_BOUND(stSettings, 1));
nUb := MIN(nUb, UPPER_BOUND(stSettings, 1));
FOR ii:= nLb TO nUb DO

	IF (stSettings[ii].stName.wsName <> "") AND (stSettings[ii].stName.wsNameId <> "")  THEN
		stSettingsView[ii].stName := stSettings[ii].stName;
		stSettingsView[ii].stGroup := stSettings[ii].stGroup;
		stSettingsView[ii].stUnit := stSettings[ii].stUnit;	
		stSettingsView[ii].stValueMin.wsName := stSettingsView[ii].stValueMin.wsNameId := TO_WSTRING(LREAL_TO_FMTSTR(REAL_TO_LREAL(stSettings[ii].fValueMin), 3, FALSE));
		stSettingsView[ii].stValueMax.wsName := stSettingsView[ii].stValueMax.wsNameId := TO_WSTRING(LREAL_TO_FMTSTR(REAL_TO_LREAL(stSettings[ii].fValueMax), 3, FALSE));	
	END_IF

	IF (stSettings[ii].stName.wsName = "") AND (stSettings[ii].stName.wsNameId = "")  THEN
		stSettingsView[ii].stDataType.wsName := "";		
	ELSIF stSettings[ii].eDataType = E_DataType.eDataType_None THEN
		stSettingsView[ii].stDataType.wsName := stSettingsView[ii].stDataType.wsNameId :="none";	
	ELSIF stSettings[ii].eDataType = E_DataType.eDataType_bool THEN
		stSettingsView[ii].stDataType.wsName := stSettingsView[ii].stDataType.wsNameId :="bool";
	ELSIF  stSettings[ii].eDataType = E_DataType.eDataType_int THEN
		stSettingsView[ii].stDataType.wsName := stSettingsView[ii].stDataType.wsNameId :="int";
	ELSIF  stSettings[ii].eDataType = E_DataType.eDataType_lreal THEN
		stSettingsView[ii].stDataType.wsName := stSettingsView[ii].stDataType.wsNameId :="lreal";
	ELSIF  stSettings[ii].eDataType = E_DataType.eDataType_time_ms THEN
		stSettingsView[ii].stDataType.wsName := stSettingsView[ii].stDataType.wsNameId :="time_ms";
	ELSIF  stSettings[ii].eDataType = E_DataType.eDataType_time_s THEN
		stSettingsView[ii].stDataType.wsName := stSettingsView[ii].stDataType.wsNameId :="time_s";	
	ELSIF  stSettings[ii].eDataType = E_DataType.eDataType_time_m THEN
		stSettingsView[ii].stDataType.wsName := stSettingsView[ii].stDataType.wsNameId :="time_m";
	ELSIF  stSettings[ii].eDataType = E_DataType.eDataType_time_h THEN
		stSettingsView[ii].stDataType.wsName := stSettingsView[ii].stDataType.wsNameId :="time_h";	
	ELSIF  stSettings[ii].eDataType = E_DataType.eDataType_wstring THEN
		stSettingsView[ii].stDataType.wsName := stSettingsView[ii].stDataType.wsNameId :="wstring";
	END_IF

	IF (stSettings[ii].stName.wsName = "") AND (stSettings[ii].stName.wsNameId = "")  THEN
		stSettingsView[ii].stRecipeMode.wsName := "";		
	ELSIF stSettings[ii].eRecipeMode = E_RecipeMode.eRecipeMode_None THEN
		stSettingsView[ii].stRecipeMode.wsName := stSettingsView[ii].stRecipeMode.wsNameId :="none";
	ELSIF  stSettings[ii].eRecipeMode = E_RecipeMode.eRecipeMode_ToFrom THEN
		stSettingsView[ii].stRecipeMode.wsName := stSettingsView[ii].stRecipeMode.wsNameId :="tofrom";
	END_IF

	IF (stSettings[ii].stName.wsName = "") AND (stSettings[ii].stName.wsNameId = "")  THEN
		stSettingsView[ii].stUserLevel.wsName := "";		
	ELSIF stSettings[ii].eUserLevel = E_User_Level.eUser_Level_none THEN
		stSettingsView[ii].stUserLevel.wsName:= stSettingsView[ii].stUserLevel.wsNameId := "none";
	ELSIF stSettings[ii].eUserLevel = E_User_Level.eUser_Level_Programmer THEN
		stSettingsView[ii].stUserLevel.wsName:= stSettingsView[ii].stUserLevel.wsNameId := "programmer";		
	ELSIF stSettings[ii].eUserLevel = E_User_Level.eUser_Level_Admin THEN
		stSettingsView[ii].stUserLevel.wsName:= stSettingsView[ii].stUserLevel.wsNameId := "admin";
	ELSIF  stSettings[ii].eUserLevel = E_User_Level.eUser_Level_Maintenance THEN
		stSettingsView[ii].stUserLevel.wsName := stSettingsView[ii].stUserLevel.wsNameId := "maintenance";
	ELSIF  stSettings[ii].eUserLevel = E_User_Level.eUser_Level_Manager THEN
		stSettingsView[ii].stUserLevel.wsName := stSettingsView[ii].stUserLevel.wsNameId := "manager";
	ELSIF  stSettings[ii].eUserLevel = E_User_Level.eUser_Level_Operator THEN
		stSettingsView[ii].stUserLevel.wsName := stSettingsView[ii].stUserLevel.wsNameId := "operator";
	ELSIF  stSettings[ii].eUserLevel = E_User_Level.eUser_Level_Level4 THEN
		stSettingsView[ii].stUserLevel.wsName := stSettingsView[ii].stUserLevel.wsNameId := "level4";
	END_IF

	IF (stSettings[ii].stName.wsName = "") AND (stSettings[ii].stName.wsNameId = "")  THEN
		stSettingsView[ii].stValue.wsName := "";		
	ELSIF stSettings[ii].eDataType = E_DataType.eDataType_bool THEN
		IF stSettings[ii].bValue THEN
			stSettingsView[ii].stValue.wsName := stSettingsView[ii].stValue.wsNameId :="true";
		ELSE
			stSettingsView[ii].stValue.wsName := stSettingsView[ii].stValue.wsNameId :="false";
		END_IF
	ELSIF stSettings[ii].eDataType = E_DataType.eDataType_int THEN
		stSettingsView[ii].stValue.wsName := TO_WSTRING(stSettings[ii].nValue);
	ELSIF stSettings[ii].eDataType = E_DataType.eDataType_lreal THEN
		stSettingsView[ii].stValue.wsName := TO_WSTRING(LREAL_TO_FMTSTR(REAL_TO_LREAL(stSettings[ii].fValue), 3, FALSE));
	ELSIF stSettings[ii].eDataType = E_DataType.eDataType_wstring THEN
		stSettingsView[ii].stValue.wsName := TO_WSTRING(stSettings[ii].sValue);
	ELSIF stSettings[ii].eDataType = E_DataType.eDataType_time_ms THEN
		stSettingsView[ii].stValue.wsName := TO_WSTRING(TO_REAL(stSettings[ii].tValue));
	ELSIF stSettings[ii].eDataType = E_DataType.eDataType_time_s THEN
		stSettingsView[ii].stValue.wsName := TO_WSTRING(TO_REAL(stSettings[ii].tValue) / 1000);	
	ELSIF stSettings[ii].eDataType = E_DataType.eDataType_time_m THEN
		stSettingsView[ii].stValue.wsName := TO_WSTRING(TO_REAL(stSettings[ii].tValue) / 60000);	
	ELSIF stSettings[ii].eDataType = E_DataType.eDataType_time_h THEN
		stSettingsView[ii].stValue.wsName := TO_WSTRING(TO_REAL(stSettings[ii].tValue) / 360000);			
	END_IF
		
END_FOR

//monitoring for control
CASE nColIndex OF

	0: // group
		IF (stSettings[nRowIndex].eDataType <> E_DataType.eDataType_None) THEN
			stControlSettingOut.bVisible_String := TRUE;
		END_IF
		
	1: // name only write by programmer
		;
		
	2: // value
		IF stSettings[nRowIndex].eDataType = E_DataType.eDataType_bool THEN
			stControlSettingOut.bVisible_Bool := TRUE;
		ELSIF stSettings[nRowIndex].eDataType = E_DataType.eDataType_int THEN
			stControlSettingOut.bVisible_Number:= TRUE;
		ELSIF stSettings[nRowIndex].eDataType = E_DataType.eDataType_lreal THEN
			stControlSettingOut.bVisible_Float:= TRUE;
		ELSIF stSettings[nRowIndex].eDataType = E_DataType.eDataType_wstring THEN
			stControlSettingOut.bVisible_String:= TRUE;
		ELSIF stSettings[nRowIndex].eDataType = E_DataType.eDataType_time_ms THEN
			stControlSettingOut.bVisible_Number:= TRUE;
		ELSIF stSettings[nRowIndex].eDataType = E_DataType.eDataType_time_s THEN
			stControlSettingOut.bVisible_Float:= TRUE;
		ELSIF stSettings[nRowIndex].eDataType = E_DataType.eDataType_time_m THEN
			stControlSettingOut.bVisible_Float:= TRUE;
		ELSIF stSettings[nRowIndex].eDataType = E_DataType.eDataType_time_h THEN
			stControlSettingOut.bVisible_Float:= TRUE;			
		ELSE
			;
		END_IF
		
	3: // min > user level programmer
		stControlSettingOut.bVisible_Float := TRUE;	
		
	4: // max > user level programmer
		stControlSettingOut.bVisible_Float := TRUE;	
		
	5: // unit only write by programmer
		;		
		
	6: // unit user level programmer
		IF (eUserLevel < E_User_Level.eUser_Level_Admin) THEN
			tofInfo.IN :=	TRUE;
			stInfo.wsName := "incorrect user level";
			stInfo.wsNameId := "incorrectuserlevel";
		ELSE
			stControlSettingOut.bVisible_UserLevel := TRUE;	
		END_IF	
		
	7: // type only write by programmer
		;
		
	8: // recipe level manager
		IF (eUserLevel < E_User_Level.eUser_Level_Manager) THEN
			tofInfo.IN :=	TRUE;
			stInfo.wsName := "incorrect user level";
			stInfo.wsNameId := "incorrectuserlevel";
		ELSE
			stControlSettingOut.bVisible_RecipeMode := TRUE;	
		END_IF	
		
END_CASE

rtSave(CLK := stControlSettingIn.stButtonSave.bClick);
IF rtSave.Q THEN
	Services.bSettingsSaved := TRUE;
	IF NOT F_ChkSettingUserLevel(eLevel := eUserLevel, stSetting := stSettings[nRowIndex], stInfo => stInfo) THEN
		tofInfo.IN :=	TRUE;
	ELSE
		CASE nColIndex OF
		
			0: // group
				IF (eUserLevel < E_User_Level.eUser_Level_Manager) 
					OR (stSettings[nRowIndex].eUserLevel = E_User_Level.eUser_Level_Programmer AND (eUserLevel <> E_User_Level.eUser_Level_Programmer))
				THEN
					tofInfo.IN :=	TRUE;
					stInfo.wsName := "incorrect user level";
					stInfo.wsNameId := "incorrectuserlevel";
				ELSE
					stSettings[nRowIndex].stGroup.wsName := stSettings[nRowIndex].stGroup.wsNameId := stControlSettingIn.wsInputString;
				END_IF
				
			1: // name only write by programmer
				;
				
			2: // value

